IF NOT _DispatchValid() THEN
	RETURN;
ELSE
	_ClearTempString();
	ZaberCommand.stringval := Tc2_Standard.CONCAT(STR1 := ZaberConfiguration.sControllerRef, STR2 := ' ');
	ZaberCommand.stringval := Tc2_Standard.CONCAT(STR1 := ZaberCommand.stringval, STR2 := Base.F_GetFirstWordInString(sInput := SUPER^._iCommandConfiguration[ZaberStatus.ZaberMethodDispatch].P_CommandConfiguration.CommandDescription));
	ZaberCommand.stringval := Tc2_Standard.CONCAT(STR1 := ZaberCommand.stringval, STR2 := ' ');
	ZaberCommand.stringval := Tc2_Standard.CONCAT(STR1 := ZaberCommand.stringval, STR2 := USINT_TO_STRING(LockstepGroup));
	ZaberCommand.stringval := Tc2_Standard.CONCAT(STR1 := ZaberCommand.stringval, STR2 := ' ');
	ZaberCommand.stringval := Tc2_Standard.CONCAT(STR1 := ZaberCommand.stringval, STR2 := F_GetAllButFirstWord(sInput := SUPER^._iCommandConfiguration[ZaberStatus.ZaberMethodDispatch].P_CommandConfiguration.CommandDescription));
	
	IF iBufferSend <> 0 AND __QUERYINTERFACE(iBufferSend, testIBufferSend) THEN
		iBufferSend.AddObject(RefObject := ZaberCommand);
	END_IF
END_IF
END_METHOD

METHOD lockstep_move_abs
VAR_INPUT
	LockstepGroup	: USINT := 1; // The address of the lockstep group must be in the range 1 to lockstep.numgroups; lockstep.numgroups: the number of lockstep groupss; Valid Values: 0 to 2
	position		: UDINT := ZaberConfiguration.SetDynamics.Position;
	max_speed 		: UDINT := ZaberConfiguration.MaxDynamics.Velocity;
	accel			: UDINT := ZaberConfiguration.MaxDynamics.Accel;
END_VAR
IF ZaberStatus.ComponentStatus.iLastCommand <> 0 THEN
	ZaberStatus.ComponentStatus.iLastCommand.P_CommandStatus.LastCommandMessage := Base.F_GetLastWordInString(__POUNAME());
END_IF

IF NOT _DispatchValid() THEN
	RETURN;
ELSE
	_ClearTempString();
	ZaberCommand.stringval := Tc2_Standard.CONCAT(STR1 := ZaberConfiguration.sControllerRef, STR2 := ' ');
	ZaberCommand.stringval := Tc2_Standard.CONCAT(STR1 := ZaberCommand.stringval, STR2 := Base.F_GetFirstWordInString(sInput := SUPER^._iCommandConfiguration[ZaberStatus.ZaberMethodDispatch].P_CommandConfiguration.CommandDescription));
	ZaberCommand.stringval := Tc2_Standard.CONCAT(STR1 := ZaberCommand.stringval, STR2 := ' ');
	ZaberCommand.stringval := Tc2_Standard.CONCAT(STR1 := ZaberCommand.stringval, STR2 := USINT_TO_STRING(LockstepGroup));
	ZaberCommand.stringval := Tc2_Standard.CONCAT(STR1 := ZaberCommand.stringval, STR2 := ' ');
	ZaberCommand.stringval := Tc2_Standard.CONCAT(STR1 := ZaberCommand.stringval, STR2 := F_GetAllButFirstWord(sInput := SUPER^._iCommandConfiguration[ZaberStatus.ZaberMethodDispatch].P_CommandConfiguration.CommandDescription));
	ZaberCommand.stringval := Tc2_Standard.CONCAT(STR1 := ZaberCommand.stringval, STR2 := ' ');
	ZaberCommand.stringval := Tc2_Standard.CONCAT(STR1 := ZaberCommand.stringval, STR2 := UDINT_TO_STRING(position));
	ZaberCommand.stringval := Tc2_Standard.CONCAT(STR1 := ZaberCommand.stringval, STR2 := ' ');
	ZaberCommand.stringval := Tc2_Standard.CONCAT(STR1 := ZaberCommand.stringval, STR2 := UDINT_TO_STRING(max_speed));
	ZaberCommand.stringval := Tc2_Standard.CONCAT(STR1 := ZaberCommand.stringval, STR2 := ' ');
	ZaberCommand.stringval := Tc2_Standard.CONCAT(STR1 := ZaberCommand.stringval, STR2 := UDINT_TO_STRING(accel));
	
	IF iBufferSend <> 0 AND __QUERYINTERFACE(iBufferSend, testIBufferSend) THEN
		iBufferSend.AddObject(RefObject := ZaberCommand);
	END_IF
END_IF
END_METHOD

METHOD lockstep_move_rel
VAR_INPUT
	LockstepGroup	: USINT := 1; // The address of the lockstep group must be in the range 1 to lockstep.numgroups; lockstep.numgroups: the number of lockstep groupss; Valid Values: 0 to 2
	distance		: UDINT := ZaberConfiguration.SetDynamics.Position - ZaberStatus.Position;
	max_speed 		: UDINT := ZaberConfiguration.MaxDynamics.Velocity;
	accel			: UDINT := ZaberConfiguration.MaxDynamics.Accel;
END_VAR
IF ZaberStatus.ComponentStatus.iLastCommand <> 0 THEN
	ZaberStatus.ComponentStatus.iLastCommand.P_CommandStatus.LastCommandMessage := Base.F_GetLastWordInString(__POUNAME());
END_IF

IF NOT _DispatchValid() THEN
	RETURN;
ELSE
	_ClearTempString();
	ZaberCommand.stringval := Tc2_Standard.CONCAT(STR1 := ZaberConfiguration.sControllerRef, STR2 := ' ');
	ZaberCommand.stringval := Tc2_Standard.CONCAT(STR1 := ZaberCommand.stringval, STR2 := Base.F_GetFirstWordInString(sInput := SUPER^._iCommandConfiguration[ZaberStatus.ZaberMethodDispatch].P_CommandConfiguration.CommandDescription));
	ZaberCommand.stringval := Tc2_Standard.CONCAT(STR1 := ZaberCommand.stringval, STR2 := ' ');
	ZaberCommand.stringval := Tc2_Standard.CONCAT(STR1 := ZaberCommand.stringval, STR2 := USINT_TO_STRING(LockstepGroup));
	ZaberCommand.stringval := Tc2_Standard.CONCAT(STR1 := ZaberCommand.stringval, STR2 := ' ');
	ZaberCommand.stringval := Tc2_Standard.CONCAT(STR1 := ZaberCommand.stringval, STR2 := F_GetAllButFirstWord(sInput := SUPER^._iCommandConfiguration[ZaberStatus.ZaberMethodDispatch].P_CommandConfiguration.CommandDescription));
	ZaberCommand.stringval := Tc2_Standard.CONCAT(STR1 := ZaberCommand.stringval, STR2 := ' ');
	ZaberCommand.stringval := Tc2_Standard.CONCAT(STR1 := ZaberCommand.stringval, STR2 := UDINT_TO_STRING(distance));
	ZaberCommand.stringval := Tc2_Standard.CONCAT(STR1 := ZaberCommand.stringval, STR2 := ' ');
	ZaberCommand.stringval := Tc2_Standard.CONCAT(STR1 := ZaberCommand.stringval, STR2 := UDINT_TO_STRING(max_speed));
	ZaberCommand.stringval := Tc2_Standard.CONCAT(STR1 := ZaberCommand.stringval, STR2 := ' ');
	ZaberCommand.stringval := Tc2_Standard.CONCAT(STR1 := ZaberCommand.stringval, STR2 := UDINT_TO_STRING(accel));
	
	IF iBufferSend <> 0 AND __QUERYINTERFACE(iBufferSend, testIBufferSend) THEN
		iBufferSend.AddObject(RefObject := ZaberCommand);
	END_IF
END_IF
END_METHOD

METHOD lockstep_move_sin_stop
VAR_INPUT
	LockstepGroup	: USINT := 1; // The address of the lockstep group must be in the range 1 to lockstep.numgroups; lockstep.numgroups: the number of lockstep groupss; Valid Values: 0 to 2
END_VAR
IF ZaberStatus.ComponentStatus.iLastCommand <> 0 THEN
	ZaberStatus.ComponentStatus.iLastCommand.P_CommandStatus.LastCommandMessage := Base.F_GetLastWordInString(__POUNAME());
END_IF

IF NOT _DispatchValid() THEN
	RETURN;
ELSE
	_ClearTempString();
	ZaberCommand.stringval := Tc2_Standard.CONCAT(STR1 := ZaberConfiguration.sControllerRef, STR2 := ' ');
	ZaberCommand.stringval := Tc2_Standard.CONCAT(STR1 := ZaberCommand.stringval, STR2 := Base.F_GetFirstWordInString(sInput := SUPER^._iCommandConfiguration[ZaberStatus.ZaberMethodDispatch].P_CommandConfiguration.CommandDescription));
	ZaberCommand.stringval := Tc2_Standard.CONCAT(STR1 := ZaberCommand.stringval, STR2 := ' ');
	ZaberCommand.stringval := Tc2_Standard.CONCAT(STR1 := ZaberCommand.stringval, STR2 := USINT_TO_STRING(LockstepGroup));
	ZaberCommand.stringval := Tc2_Standard.CONCAT(STR1 := ZaberCommand.stringval, STR2 := ' ');
	ZaberCommand.stringval := Tc2_Standard.CONCAT(STR1 := ZaberCommand.stringval, STR2 := F_GetAllButFirstWord(sInput := SUPER^._iCommandConfiguration[ZaberStatus.ZaberMethodDispatch].P_CommandConfiguration.CommandDescription));
	
	IF iBufferSend <> 0 AND __QUERYINTERFACE(iBufferSend, testIBufferSend) THEN
		iBufferSend.AddObject(RefObject := ZaberCommand);
	END_IF
END_IF
END_METHOD

METHOD lockstep_move_stored
IF ZaberStatus.ComponentStatus.iLastCommand <> 0 THEN
	ZaberStatus.ComponentStatus.iLastCommand.P_CommandStatus.LastCommandMessage := Base.F_GetLastWordInString(__POUNAME());
END_IF

IF NOT _DispatchValid() THEN
	RETURN;
ELSE
	_BuildCommandStringNoArgs();
	
	IF iBufferSend <> 0 AND __QUERYINTERFACE(iBufferSend, testIBufferSend) THEN
		iBufferSend.AddObject(RefObject := ZaberCommand);
	END_IF
END_IF
END_METHOD

METHOD lockstep_move_vel
VAR_INPUT
	LockstepGroup	: USINT := 1; // The address of the lockstep group must be in the range 1 to lockstep.numgroups; lockstep.numgroups: the number of lockstep groupss; Valid Values: 0 to 2
	velocity		: DINT := ZaberConfiguration.SetDynamics.Velocity;
	accel			: UDINT := ZaberConfiguration.MaxDynamics.Accel;
END_VAR
IF ZaberStatus.ComponentStatus.iLastCommand <> 0 THEN
	ZaberStatus.ComponentStatus.iLastCommand.P_CommandStatus.LastCommandMessage := Base.F_GetLastWordInString(__POUNAME());
END_IF

IF NOT _DispatchValid() THEN
	RETURN;
ELSE
	_ClearTempString();
	ZaberCommand.stringval := Tc2_Standard.CONCAT(STR1 := ZaberConfiguration.sControllerRef, STR2 := ' ');
	ZaberCommand.stringval := Tc2_Standard.CONCAT(STR1 := ZaberCommand.stringval, STR2 := Base.F_GetFirstWordInString(sInput := SUPER^._iCommandConfiguration[ZaberStatus.ZaberMethodDispatch].P_CommandConfiguration.CommandDescription));
	ZaberCommand.stringval := Tc2_Standard.CONCAT(STR1 := ZaberCommand.stringval, STR2 := ' ');
	ZaberCommand.stringval := Tc2_Standard.CONCAT(STR1 := ZaberCommand.stringval, STR2 := USINT_TO_STRING(LockstepGroup));
	ZaberCommand.stringval := Tc2_Standard.CONCAT(STR1 := ZaberCommand.stringval, STR2 := ' ');
	ZaberCommand.stringval := Tc2_Standard.CONCAT(STR1 := ZaberCommand.stringval, STR2 := F_GetAllButFirstWord(sInput := SUPER^._iCommandConfiguration[ZaberStatus.ZaberMethodDispatch].P_CommandConfiguration.CommandDescription));
	ZaberCommand.stringval := Tc2_Standard.CONCAT(STR1 := ZaberCommand.stringval, STR2 := ' ');
	ZaberCommand.stringval := Tc2_Standard.CONCAT(STR1 := ZaberCommand.stringval, STR2 := UDINT_TO_STRING(velocity));
	ZaberCommand.stringval := Tc2_Standard.CONCAT(STR1 := ZaberCommand.stringval, STR2 := ' ');
	ZaberCommand.stringval := Tc2_Standard.CONCAT(STR1 := ZaberCommand.stringval, STR2 := UDINT_TO_STRING(accel));
	
	IF iBufferSend <> 0 AND __QUERYINTERFACE(iBufferSend, testIBufferSend) THEN
		iBufferSend.AddObject(RefObject := ZaberCommand);
	END_IF
END_IF
END_METHOD

METHOD lockstep_park
VAR_INPUT
	LockstepGroup	: USINT := 1; // The address of the lockstep group must be in the range 1 to lockstep.numgroups; lockstep.numgroups: the number of lockstep groupss; Valid Values: 0 to 2
END_VAR
IF ZaberStatus.ComponentStatus.iLastCommand <> 0 THEN
	ZaberStatus.ComponentStatus.iLastCommand.P_CommandStatus.LastCommandMessage := Base.F_GetLastWordInString(__POUNAME());
END_IF

IF NOT _DispatchValid() THEN
	RETURN;
ELSE
	_ClearTempString();
	ZaberCommand.stringval := Tc2_Standard.CONCAT(STR1 := ZaberConfiguration.sControllerRef, STR2 := ' ');
	ZaberCommand.stringval := Tc2_Standard.CONCAT(STR1 := ZaberCommand.stringval, STR2 := Base.F_GetFirstWordInString(sInput := SUPER^._iCommandConfiguration[ZaberStatus.ZaberMethodDispatch].P_CommandConfiguration.CommandDescription));
	ZaberCommand.stringval := Tc2_Standard.CONCAT(STR1 := ZaberCommand.stringval, STR2 := ' ');
	ZaberCommand.stringval := Tc2_Standard.CONCAT(STR1 := ZaberCommand.stringval, STR2 := USINT_TO_STRING(LockstepGroup));
	ZaberCommand.stringval := Tc2_Standard.CONCAT(STR1 := ZaberCommand.stringval, STR2 := ' ');
	ZaberCommand.stringval := Tc2_Standard.CONCAT(STR1 := ZaberCommand.stringval, STR2 := F_GetAllButFirstWord(sInput := SUPER^._iCommandConfiguration[ZaberStatus.ZaberMethodDispatch].P_CommandConfiguration.CommandDescription));
	
	IF iBufferSend <> 0 AND __QUERYINTERFACE(iBufferSend, testIBufferSend) THEN
		iBufferSend.AddObject(RefObject := ZaberCommand);
	END_IF
END_IF
END_METHOD

METHOD lockstep_print
VAR_INPUT
	LockstepGroup	: USINT := 1; // The address of the lockstep group must be in the range 1 to lockstep.numgroups; lockstep.numgroups: the number of lockstep groupss; Valid Values: 0 to 2
END_VAR
IF ZaberStatus.ComponentStatus.iLastCommand <> 0 THEN
	ZaberStatus.ComponentStatus.iLastCommand.P_CommandStatus.LastCommandMessage := Base.F_GetLastWordInString(__POUNAME());
END_IF

IF NOT _DispatchValid() THEN
	RETURN;
ELSE
	_ClearTempString();
	ZaberCommand.stringval := Tc2_Standard.CONCAT(STR1 := ZaberConfiguration.sControllerRef, STR2 := ' ');
	ZaberCommand.stringval := Tc2_Standard.CONCAT(STR1 := ZaberCommand.stringval, STR2 := Base.F_GetFirstWordInString(sInput := SUPER^._iCommandConfiguration[ZaberStatus.ZaberMethodDispatch].P_CommandConfiguration.CommandDescription));
	ZaberCommand.stringval := Tc2_Standard.CONCAT(STR1 := ZaberCommand.stringval, STR2 := ' ');
	ZaberCommand.stringval := Tc2_Standard.CONCAT(STR1 := ZaberCommand.stringval, STR2 := USINT_TO_STRING(LockstepGroup));
	ZaberCommand.stringval := Tc2_Standard.CONCAT(STR1 := ZaberCommand.stringval, STR2 := ' ');
	ZaberCommand.stringval := Tc2_Standard.CONCAT(STR1 := ZaberCommand.stringval, STR2 := F_GetAllButFirstWord(sInput := SUPER^._iCommandConfiguration[ZaberStatus.ZaberMethodDispatch].P_CommandConfiguration.CommandDescription));
	
	IF iBufferSend <> 0 AND __QUERYINTERFACE(iBufferSend, testIBufferSend) THEN
		iBufferSend.AddObject(RefObject := ZaberCommand);
	END_IF
END_IF
END_METHOD

METHOD lockstep_set_tolerance
VAR_INPUT
	LockstepGroup	: USINT := 1; // The address of the lockstep group must be in the range 1 to lockstep.numgroups; lockstep.numgroups: the number of lockstep groupss; Valid Values: 0 to 2
	Tolerance 		: UDINT := 150;
END_VAR
IF ZaberStatus.ComponentStatus.iLastCommand <> 0 THEN
	ZaberStatus.ComponentStatus.iLastCommand.P_CommandStatus.LastCommandMessage := Base.F_GetLastWordInString(__POUNAME());
END_IF

IF NOT _DispatchValid() THEN
	RETURN;
ELSE
	_ClearTempString();
	ZaberCommand.stringval := Tc2_Standard.CONCAT(STR1 := ZaberConfiguration.sControllerRef, STR2 := ' ');
	ZaberCommand.stringval := Tc2_Standard.CONCAT(STR1 := ZaberCommand.stringval, STR2 := UINT_TO_STRING(ZaberConfiguration.AxisRef));
	ZaberCommand.stringval := Tc2_Standard.CONCAT(STR1 := ZaberCommand.stringval, STR2 := ' ');
	ZaberCommand.stringval := Tc2_Standard.CONCAT(STR1 := ZaberCommand.stringval, STR2 := Base.F_GetFirstWordInString(sInput := SUPER^._iCommandConfiguration[ZaberStatus.ZaberMethodDispatch].P_CommandConfiguration.CommandDescription));
	ZaberCommand.stringval := Tc2_Standard.CONCAT(STR1 := ZaberCommand.stringval, STR2 := ' ');
	ZaberCommand.stringval := Tc2_Standard.CONCAT(STR1 := ZaberCommand.stringval, STR2 := USINT_TO_STRING(LockstepGroup));
	ZaberCommand.stringval := Tc2_Standard.CONCAT(STR1 := ZaberCommand.stringval, STR2 := ' ');
	ZaberCommand.stringval := Tc2_Standard.CONCAT(STR1 := ZaberCommand.stringval, STR2 := F_GetAllButFirstWord(sInput := SUPER^._iCommandConfiguration[ZaberStatus.ZaberMethodDispatch].P_CommandConfiguration.CommandDescription));
	ZaberCommand.stringval := Tc2_Standard.CONCAT(STR1 := ZaberCommand.stringval, STR2 := ' ');
	ZaberCommand.stringval := Tc2_Standard.CONCAT(STR1 := ZaberCommand.stringval, STR2 := UDINT_TO_STRING(Tolerance));;
	
	IF iBufferSend <> 0 AND __QUERYINTERFACE(iBufferSend, testIBufferSend) THEN
		iBufferSend.AddObject(RefObject := ZaberCommand);
	END_IF
END_IF
END_METHOD

METHOD lockstep_setup_disable
VAR_INPUT
	LockstepGroup	: USINT := 1; // The address of the lockstep group must be in the range 1 to lockstep.numgroups; lockstep.numgroups: the number of lockstep groupss; Valid Values: 0 to 2
END_VAR
IF ZaberStatus.ComponentStatus.iLastCommand <> 0 THEN
	ZaberStatus.ComponentStatus.iLastCommand.P_CommandStatus.LastCommandMessage := Base.F_GetLastWordInString(__POUNAME());
END_IF

IF NOT _DispatchValid() THEN
	RETURN;
ELSE
	_ClearTempString();
	ZaberCommand.stringval := Tc2_Standard.CONCAT(STR1 := ZaberConfiguration.sControllerRef, STR2 := ' ');
	ZaberCommand.stringval := Tc2_Standard.CONCAT(STR1 := ZaberCommand.stringval, STR2 := UINT_TO_STRING(ZaberConfiguration.AxisRef));
	ZaberCommand.stringval := Tc2_Standard.CONCAT(STR1 := ZaberCommand.stringval, STR2 := ' ');
	ZaberCommand.stringval := Tc2_Standard.CONCAT(STR1 := ZaberCommand.stringval, STR2 := Base.F_GetFirstWordInString(sInput := SUPER^._iCommandConfiguration[ZaberStatus.ZaberMethodDispatch].P_CommandConfiguration.CommandDescription));
	ZaberCommand.stringval := Tc2_Standard.CONCAT(STR1 := ZaberCommand.stringval, STR2 := ' ');
	ZaberCommand.stringval := Tc2_Standard.CONCAT(STR1 := ZaberCommand.stringval, STR2 := USINT_TO_STRING(LockstepGroup));
	ZaberCommand.stringval := Tc2_Standard.CONCAT(STR1 := ZaberCommand.stringval, STR2 := ' ');
	ZaberCommand.stringval := Tc2_Standard.CONCAT(STR1 := ZaberCommand.stringval, STR2 := F_GetAllButFirstWord(sInput := SUPER^._iCommandConfiguration[ZaberStatus.ZaberMethodDispatch].P_CommandConfiguration.CommandDescription));
	
	IF iBufferSend <> 0 AND __QUERYINTERFACE(iBufferSend, testIBufferSend) THEN
		iBufferSend.AddObject(RefObject := ZaberCommand);
	END_IF
END_IF
END_METHOD

METHOD lockstep_setup_enable
VAR_INPUT
	LockstepGroup	: USINT := 1; // The address of the lockstep group must be in the range 1 to lockstep.numgroups; lockstep.numgroups: the number of lockstep groupss; Valid Values: 0 to 2
	PrimaryAxis 	: USINT := 1;
	SecondaryAxis	: USINT := 2;
END_VAR
IF ZaberStatus.ComponentStatus.iLastCommand <> 0 THEN
	ZaberStatus.ComponentStatus.iLastCommand.P_CommandStatus.LastCommandMessage := Base.F_GetLastWordInString(__POUNAME());
END_IF

IF NOT _DispatchValid() THEN
	RETURN;
ELSE
	_ClearTempString();
	ZaberCommand.stringval := Tc2_Standard.CONCAT(STR1 := ZaberConfiguration.sControllerRef, STR2 := ' ');
	ZaberCommand.stringval := Tc2_Standard.CONCAT(STR1 := ZaberCommand.stringval, STR2 := UINT_TO_STRING(ZaberConfiguration.AxisRef));
	ZaberCommand.stringval := Tc2_Standard.CONCAT(STR1 := ZaberCommand.stringval, STR2 := ' ');
	ZaberCommand.stringval := Tc2_Standard.CONCAT(STR1 := ZaberCommand.stringval, STR2 := Base.F_GetFirstWordInString(sInput := SUPER^._iCommandConfiguration[ZaberStatus.ZaberMethodDispatch].P_CommandConfiguration.CommandDescription));
	ZaberCommand.stringval := Tc2_Standard.CONCAT(STR1 := ZaberCommand.stringval, STR2 := ' ');
	ZaberCommand.stringval := Tc2_Standard.CONCAT(STR1 := ZaberCommand.stringval, STR2 := USINT_TO_STRING(LockstepGroup));
	ZaberCommand.stringval := Tc2_Standard.CONCAT(STR1 := ZaberCommand.stringval, STR2 := ' ');
	ZaberCommand.stringval := Tc2_Standard.CONCAT(STR1 := ZaberCommand.stringval, STR2 := F_GetAllButFirstWord(sInput := SUPER^._iCommandConfiguration[ZaberStatus.ZaberMethodDispatch].P_CommandConfiguration.CommandDescription));
	ZaberCommand.stringval := Tc2_Standard.CONCAT(STR1 := ZaberCommand.stringval, STR2 := ' ');
	ZaberCommand.stringval := Tc2_Standard.CONCAT(STR1 := ZaberCommand.stringval, STR2 := USINT_TO_STRING(PrimaryAxis));
	ZaberCommand.stringval := Tc2_Standard.CONCAT(STR1 := ZaberCommand.stringval, STR2 := ' ');
	ZaberCommand.stringval := Tc2_Standard.CONCAT(STR1 := ZaberCommand.stringval, STR2 := USINT_TO_STRING(SecondaryAxis));
	
	IF iBufferSend <> 0 AND __QUERYINTERFACE(iBufferSend, testIBufferSend) THEN
		iBufferSend.AddObject(RefObject := ZaberCommand);
	END_IF
END_IF
END_METHOD

METHOD lockstep_stop
VAR_INPUT
	LockstepGroup	: USINT := 1; // The address of the lockstep group must be in the range 1 to lockstep.numgroups; lockstep.numgroups: the number of lockstep groupss; Valid Values: 0 to 2
END_VAR
IF ZaberStatus.ComponentStatus.iLastCommand <> 0 THEN
	ZaberStatus.ComponentStatus.iLastCommand.P_CommandStatus.LastCommandMessage := Base.F_GetLastWordInString(__POUNAME());
END_IF

IF NOT _DispatchValid() THEN
	RETURN;
ELSE
	_ClearTempString();
	ZaberCommand.stringval := Tc2_Standard.CONCAT(STR1 := ZaberConfiguration.sControllerRef, STR2 := ' ');
	ZaberCommand.stringval := Tc2_Standard.CONCAT(STR1 := ZaberCommand.stringval, STR2 := UINT_TO_STRING(ZaberConfiguration.AxisRef));
	ZaberCommand.stringval := Tc2_Standard.CONCAT(STR1 := ZaberCommand.stringval, STR2 := ' ');
	ZaberCommand.stringval := Tc2_Standard.CONCAT(STR1 := ZaberCommand.stringval, STR2 := Base.F_GetFirstWordInString(sInput := SUPER^._iCommandConfiguration[ZaberStatus.ZaberMethodDispatch].P_CommandConfiguration.CommandDescription));
	ZaberCommand.stringval := Tc2_Standard.CONCAT(STR1 := ZaberCommand.stringval, STR2 := ' ');
	ZaberCommand.stringval := Tc2_Standard.CONCAT(STR1 := ZaberCommand.stringval, STR2 := USINT_TO_STRING(LockstepGroup));
	ZaberCommand.stringval := Tc2_Standard.CONCAT(STR1 := ZaberCommand.stringval, STR2 := ' ');
	ZaberCommand.stringval := Tc2_Standard.CONCAT(STR1 := ZaberCommand.stringval, STR2 := F_GetAllButFirstWord(sInput := SUPER^._iCommandConfiguration[ZaberStatus.ZaberMethodDispatch].P_CommandConfiguration.CommandDescription));
	
	IF iBufferSend <> 0 AND __QUERYINTERFACE(iBufferSend, testIBufferSend) THEN
		iBufferSend.AddObject(RefObject := ZaberCommand);
	END_IF
END_IF
END_METHOD

METHOD lockstep_unpark
VAR_INPUT
	LockstepGroup	: USINT := 1; // The address of the lockstep group must be in the range 1 to lockstep.numgroups; lockstep.numgroups: the number of lockstep groupss; Valid Values: 0 to 2
END_VAR
IF ZaberStatus.ComponentStatus.iLastCommand <> 0 THEN
	ZaberStatus.ComponentStatus.iLastCommand.P_CommandStatus.LastCommandMessage := Base.F_GetLastWordInString(__POUNAME());
END_IF

IF NOT _DispatchValid() THEN
	RETURN;
ELSE
	_ClearTempString();
	ZaberCommand.stringval := Tc2_Standard.CONCAT(STR1 := ZaberConfiguration.sControllerRef, STR2 := ' ');
	ZaberCommand.stringval := Tc2_Standard.CONCAT(STR1 := ZaberCommand.stringval, STR2 := UINT_TO_STRING(ZaberConfiguration.AxisRef));
	ZaberCommand.stringval := Tc2_Standard.CONCAT(STR1 := ZaberCommand.stringval, STR2 := ' ');
	ZaberCommand.stringval := Tc2_Standard.CONCAT(STR1 := ZaberCommand.stringval, STR2 := Base.F_GetFirstWordInString(sInput := SUPER^._iCommandConfiguration[ZaberStatus.ZaberMethodDispatch].P_CommandConfiguration.CommandDescription));
	ZaberCommand.stringval := Tc2_Standard.CONCAT(STR1 := ZaberCommand.stringval, STR2 := ' ');
	ZaberCommand.stringval := Tc2_Standard.CONCAT(STR1 := ZaberCommand.stringval, STR2 := USINT_TO_STRING(LockstepGroup));
	ZaberCommand.stringval := Tc2_Standard.CONCAT(STR1 := ZaberCommand.stringval, STR2 := ' ');
	ZaberCommand.stringval := Tc2_Standard.CONCAT(STR1 := ZaberCommand.stringval, STR2 := F_GetAllButFirstWord(sInput := SUPER^._iCommandConfiguration[ZaberStatus.ZaberMethodDispatch].P_CommandConfiguration.CommandDescription));
	
	IF iBufferSend <> 0 AND __QUERYINTERFACE(iBufferSend, testIBufferSend) THEN
		iBufferSend.AddObject(RefObject := ZaberCommand);
	END_IF
END_IF
END_METHOD

METHOD move_index
IF ZaberStatus.ComponentStatus.iLastCommand <> 0 THEN
	ZaberStatus.ComponentStatus.iLastCommand.P_CommandStatus.LastCommandMessage := Base.F_GetLastWordInString(__POUNAME());
END_IF

IF NOT _DispatchValid() THEN
	RETURN;
ELSE
	_BuildCommandStringNoArgs();
	
	IF iBufferSend <> 0 AND __QUERYINTERFACE(iBufferSend, testIBufferSend) THEN
		iBufferSend.AddObject(RefObject := ZaberCommand);
	END_IF
END_IF
END_METHOD

METHOD move_rel
VAR_INPUT
	distance		: UDINT;
	max_speed 		: UDINT;
	accel			: UDINT;
END_VAR
IF ZaberStatus.ComponentStatus.iLastCommand <> 0 THEN
	ZaberStatus.ComponentStatus.iLastCommand.P_CommandStatus.LastCommandMessage := Base.F_GetLastWordInString(__POUNAME());
END_IF

IF NOT _DispatchValid() THEN
	RETURN;
ELSE
	_ClearTempString();
	ZaberCommand.stringval := Tc2_Standard.CONCAT(STR1 := ZaberConfiguration.sControllerRef, STR2 := ' ');
	ZaberCommand.stringval := Tc2_Standard.CONCAT(STR1 := ZaberCommand.stringval, STR2 := UINT_TO_STRING(ZaberConfiguration.AxisRef));
	ZaberCommand.stringval := Tc2_Standard.CONCAT(STR1 := ZaberCommand.stringval, STR2 := ' ');
	ZaberCommand.stringval := Tc2_Standard.CONCAT(STR1 := ZaberCommand.stringval, STR2 := SUPER^._iCommandConfiguration[ZaberStatus.ZaberMethodDispatch].P_CommandConfiguration.CommandDescription);
	ZaberCommand.stringval := Tc2_Standard.CONCAT(STR1 := ZaberCommand.stringval, STR2 := ' ');
	ZaberCommand.stringval := Tc2_Standard.CONCAT(STR1 := ZaberCommand.stringval, STR2 := UDINT_TO_STRING(distance));
	ZaberCommand.stringval := Tc2_Standard.CONCAT(STR1 := ZaberCommand.stringval, STR2 := ' ');
	ZaberCommand.stringval := Tc2_Standard.CONCAT(STR1 := ZaberCommand.stringval, STR2 := UDINT_TO_STRING(max_speed));
	ZaberCommand.stringval := Tc2_Standard.CONCAT(STR1 := ZaberCommand.stringval, STR2 := ' ');
	ZaberCommand.stringval := Tc2_Standard.CONCAT(STR1 := ZaberCommand.stringval, STR2 := UDINT_TO_STRING(accel));
		
	IF iBufferSend <> 0 AND __QUERYINTERFACE(iBufferSend, testIBufferSend) THEN
		iBufferSend.AddObject(RefObject := ZaberCommand);
	END_IF
END_IF
END_METHOD

METHOD move_sin_stop
IF ZaberStatus.ComponentStatus.iLastCommand <> 0 THEN
	ZaberStatus.ComponentStatus.iLastCommand.P_CommandStatus.LastCommandMessage := Base.F_GetLastWordInString(__POUNAME());
END_IF

IF NOT _DispatchValid() THEN
	RETURN;
ELSE
	_ClearTempString();
	ZaberCommand.stringval := Tc2_Standard.CONCAT(STR1 := ZaberConfiguration.sControllerRef, STR2 := ' ');
	ZaberCommand.stringval := Tc2_Standard.CONCAT(STR1 := ZaberCommand.stringval, STR2 := UINT_TO_STRING(ZaberConfiguration.AxisRef));
	ZaberCommand.stringval := Tc2_Standard.CONCAT(STR1 := ZaberCommand.stringval, STR2 := ' ');
	ZaberCommand.stringval := Tc2_Standard.CONCAT(STR1 := ZaberCommand.stringval, STR2 := SUPER^._iCommandConfiguration[ZaberStatus.ZaberMethodDispatch].P_CommandConfiguration.CommandDescription);
	
	IF iBufferSend <> 0 AND __QUERYINTERFACE(iBufferSend, testIBufferSend) THEN
		iBufferSend.AddObject(RefObject := ZaberCommand);
	END_IF
END_IF
END_METHOD

METHOD move_stored
IF ZaberStatus.ComponentStatus.iLastCommand <> 0 THEN
	ZaberStatus.ComponentStatus.iLastCommand.P_CommandStatus.LastCommandMessage := Base.F_GetLastWordInString(__POUNAME());
END_IF

IF NOT _DispatchValid() THEN
	RETURN;
ELSE
	_BuildCommandStringNoArgs();
	
	IF iBufferSend <> 0 AND __QUERYINTERFACE(iBufferSend, testIBufferSend) THEN
		iBufferSend.AddObject(RefObject := ZaberCommand);
	END_IF
END_IF
END_METHOD

METHOD pvt_buffer_erase
IF ZaberStatus.ComponentStatus.iLastCommand <> 0 THEN
	ZaberStatus.ComponentStatus.iLastCommand.P_CommandStatus.LastCommandMessage := Base.F_GetLastWordInString(__POUNAME());
END_IF

IF NOT _DispatchValid() THEN
	RETURN;
ELSE
	_BuildCommandStringNoArgs();
	
	IF iBufferSend <> 0 AND __QUERYINTERFACE(iBufferSend, testIBufferSend) THEN
		iBufferSend.AddObject(RefObject := ZaberCommand);
	END_IF
END_IF
END_METHOD

METHOD pvt_buffer_print
IF ZaberStatus.ComponentStatus.iLastCommand <> 0 THEN
	ZaberStatus.ComponentStatus.iLastCommand.P_CommandStatus.LastCommandMessage := Base.F_GetLastWordInString(__POUNAME());
END_IF

IF NOT _DispatchValid() THEN
	RETURN;
ELSE
	_BuildCommandStringNoArgs();
	
	IF iBufferSend <> 0 AND __QUERYINTERFACE(iBufferSend, testIBufferSend) THEN
		iBufferSend.AddObject(RefObject := ZaberCommand);
	END_IF
END_IF
END_METHOD

METHOD pvt_call
IF ZaberStatus.ComponentStatus.iLastCommand <> 0 THEN
	ZaberStatus.ComponentStatus.iLastCommand.P_CommandStatus.LastCommandMessage := Base.F_GetLastWordInString(__POUNAME());
END_IF

IF NOT _DispatchValid() THEN
	RETURN;
ELSE
	_BuildCommandStringNoArgs();
	
	IF iBufferSend <> 0 AND __QUERYINTERFACE(iBufferSend, testIBufferSend) THEN
		iBufferSend.AddObject(RefObject := ZaberCommand);
	END_IF
END_IF
END_METHOD

METHOD pvt_fifo
IF ZaberStatus.ComponentStatus.iLastCommand <> 0 THEN
	ZaberStatus.ComponentStatus.iLastCommand.P_CommandStatus.LastCommandMessage := Base.F_GetLastWordInString(__POUNAME());
END_IF

IF NOT _DispatchValid() THEN
	RETURN;
ELSE
	_BuildCommandStringNoArgs();
	
	IF iBufferSend <> 0 AND __QUERYINTERFACE(iBufferSend, testIBufferSend) THEN
		iBufferSend.AddObject(RefObject := ZaberCommand);
	END_IF
END_IF
END_METHOD

METHOD pvt_info
IF ZaberStatus.ComponentStatus.iLastCommand <> 0 THEN
	ZaberStatus.ComponentStatus.iLastCommand.P_CommandStatus.LastCommandMessage := Base.F_GetLastWordInString(__POUNAME());
END_IF

IF NOT _DispatchValid() THEN
	RETURN;
ELSE
	_BuildCommandStringNoArgs();
	
	IF iBufferSend <> 0 AND __QUERYINTERFACE(iBufferSend, testIBufferSend) THEN
		iBufferSend.AddObject(RefObject := ZaberCommand);
	END_IF
END_IF
END_METHOD

METHOD pvt_io_cancel_schedule
IF ZaberStatus.ComponentStatus.iLastCommand <> 0 THEN
	ZaberStatus.ComponentStatus.iLastCommand.P_CommandStatus.LastCommandMessage := Base.F_GetLastWordInString(__POUNAME());
END_IF

IF NOT _DispatchValid() THEN
	RETURN;
ELSE
	_BuildCommandStringNoArgs();
	
	IF iBufferSend <> 0 AND __QUERYINTERFACE(iBufferSend, testIBufferSend) THEN
		iBufferSend.AddObject(RefObject := ZaberCommand);
	END_IF
END_IF
END_METHOD

METHOD pvt_io_set_ao
IF ZaberStatus.ComponentStatus.iLastCommand <> 0 THEN
	ZaberStatus.ComponentStatus.iLastCommand.P_CommandStatus.LastCommandMessage := Base.F_GetLastWordInString(__POUNAME());
END_IF

IF NOT _DispatchValid() THEN
	RETURN;
ELSE
	_BuildCommandStringNoArgs();
	
	IF iBufferSend <> 0 AND __QUERYINTERFACE(iBufferSend, testIBufferSend) THEN
		iBufferSend.AddObject(RefObject := ZaberCommand);
	END_IF
END_IF
END_METHOD

METHOD pvt_io_set_ao_schedule
IF ZaberStatus.ComponentStatus.iLastCommand <> 0 THEN
	ZaberStatus.ComponentStatus.iLastCommand.P_CommandStatus.LastCommandMessage := Base.F_GetLastWordInString(__POUNAME());
END_IF

IF NOT _DispatchValid() THEN
	RETURN;
ELSE
	_BuildCommandStringNoArgs();
	
	IF iBufferSend <> 0 AND __QUERYINTERFACE(iBufferSend, testIBufferSend) THEN
		iBufferSend.AddObject(RefObject := ZaberCommand);
	END_IF
END_IF
END_METHOD

METHOD pvt_io_set_do
IF ZaberStatus.ComponentStatus.iLastCommand <> 0 THEN
	ZaberStatus.ComponentStatus.iLastCommand.P_CommandStatus.LastCommandMessage := Base.F_GetLastWordInString(__POUNAME());
END_IF

IF NOT _DispatchValid() THEN
	RETURN;
ELSE
	_BuildCommandStringNoArgs();
	
	IF iBufferSend <> 0 AND __QUERYINTERFACE(iBufferSend, testIBufferSend) THEN
		iBufferSend.AddObject(RefObject := ZaberCommand);
	END_IF
END_IF
END_METHOD

METHOD pvt_io_set_do_schedule
IF ZaberStatus.ComponentStatus.iLastCommand <> 0 THEN
	ZaberStatus.ComponentStatus.iLastCommand.P_CommandStatus.LastCommandMessage := Base.F_GetLastWordInString(__POUNAME());
END_IF

IF NOT _DispatchValid() THEN
	RETURN;
ELSE
	_BuildCommandStringNoArgs();
	
	IF iBufferSend <> 0 AND __QUERYINTERFACE(iBufferSend, testIBufferSend) THEN
		iBufferSend.AddObject(RefObject := ZaberCommand);
	END_IF
END_IF
END_METHOD

METHOD pvt_point
IF ZaberStatus.ComponentStatus.iLastCommand <> 0 THEN
	ZaberStatus.ComponentStatus.iLastCommand.P_CommandStatus.LastCommandMessage := Base.F_GetLastWordInString(__POUNAME());
END_IF

IF NOT _DispatchValid() THEN
	RETURN;
ELSE
	_BuildCommandStringNoArgs();
	
	IF iBufferSend <> 0 AND __QUERYINTERFACE(iBufferSend, testIBufferSend) THEN
		iBufferSend.AddObject(RefObject := ZaberCommand);
	END_IF
END_IF
END_METHOD

METHOD pvt_setup_disable
IF ZaberStatus.ComponentStatus.iLastCommand <> 0 THEN
	ZaberStatus.ComponentStatus.iLastCommand.P_CommandStatus.LastCommandMessage := Base.F_GetLastWordInString(__POUNAME());
END_IF

IF NOT _DispatchValid() THEN
	RETURN;
ELSE
	_BuildCommandStringNoArgs();
	
	IF iBufferSend <> 0 AND __QUERYINTERFACE(iBufferSend, testIBufferSend) THEN
		iBufferSend.AddObject(RefObject := ZaberCommand);
	END_IF
END_IF
END_METHOD

METHOD pvt_setup_live
IF ZaberStatus.ComponentStatus.iLastCommand <> 0 THEN
	ZaberStatus.ComponentStatus.iLastCommand.P_CommandStatus.LastCommandMessage := Base.F_GetLastWordInString(__POUNAME());
END_IF

IF NOT _DispatchValid() THEN
	RETURN;
ELSE
	_BuildCommandStringNoArgs();
	
	IF iBufferSend <> 0 AND __QUERYINTERFACE(iBufferSend, testIBufferSend) THEN
		iBufferSend.AddObject(RefObject := ZaberCommand);
	END_IF
END_IF
END_METHOD

METHOD pvt_setup_store
IF ZaberStatus.ComponentStatus.iLastCommand <> 0 THEN
	ZaberStatus.ComponentStatus.iLastCommand.P_CommandStatus.LastCommandMessage := Base.F_GetLastWordInString(__POUNAME());
END_IF

IF NOT _DispatchValid() THEN
	RETURN;
ELSE
	_BuildCommandStringNoArgs();
	
	IF iBufferSend <> 0 AND __QUERYINTERFACE(iBufferSend, testIBufferSend) THEN
		iBufferSend.AddObject(RefObject := ZaberCommand);
	END_IF
END_IF
END_METHOD

METHOD scope_add
IF ZaberStatus.ComponentStatus.iLastCommand <> 0 THEN
	ZaberStatus.ComponentStatus.iLastCommand.P_CommandStatus.LastCommandMessage := Base.F_GetLastWordInString(__POUNAME());
END_IF

IF NOT _DispatchValid() THEN
	RETURN;
ELSE
	_BuildCommandStringNoArgs();
	
	IF iBufferSend <> 0 AND __QUERYINTERFACE(iBufferSend, testIBufferSend) THEN
		iBufferSend.AddObject(RefObject := ZaberCommand);
	END_IF
END_IF
END_METHOD

METHOD scope_add_io_ai
IF ZaberStatus.ComponentStatus.iLastCommand <> 0 THEN
	ZaberStatus.ComponentStatus.iLastCommand.P_CommandStatus.LastCommandMessage := Base.F_GetLastWordInString(__POUNAME());
END_IF

IF NOT _DispatchValid() THEN
	RETURN;
ELSE
	_BuildCommandStringNoArgs();
	
	IF iBufferSend <> 0 AND __QUERYINTERFACE(iBufferSend, testIBufferSend) THEN
		iBufferSend.AddObject(RefObject := ZaberCommand);
	END_IF
END_IF
END_METHOD

METHOD scope_add_io_ao
IF ZaberStatus.ComponentStatus.iLastCommand <> 0 THEN
	ZaberStatus.ComponentStatus.iLastCommand.P_CommandStatus.LastCommandMessage := Base.F_GetLastWordInString(__POUNAME());
END_IF

IF NOT _DispatchValid() THEN
	RETURN;
ELSE
	_BuildCommandStringNoArgs();
	
	IF iBufferSend <> 0 AND __QUERYINTERFACE(iBufferSend, testIBufferSend) THEN
		iBufferSend.AddObject(RefObject := ZaberCommand);
	END_IF
END_IF
END_METHOD

METHOD scope_add_io_di
IF ZaberStatus.ComponentStatus.iLastCommand <> 0 THEN
	ZaberStatus.ComponentStatus.iLastCommand.P_CommandStatus.LastCommandMessage := Base.F_GetLastWordInString(__POUNAME());
END_IF

IF NOT _DispatchValid() THEN
	RETURN;
ELSE
	_BuildCommandStringNoArgs();
	
	IF iBufferSend <> 0 AND __QUERYINTERFACE(iBufferSend, testIBufferSend) THEN
		iBufferSend.AddObject(RefObject := ZaberCommand);
	END_IF
END_IF
END_METHOD

METHOD scope_add_io_do
IF ZaberStatus.ComponentStatus.iLastCommand <> 0 THEN
	ZaberStatus.ComponentStatus.iLastCommand.P_CommandStatus.LastCommandMessage := Base.F_GetLastWordInString(__POUNAME());
END_IF

IF NOT _DispatchValid() THEN
	RETURN;
ELSE
	_BuildCommandStringNoArgs();
	
	IF iBufferSend <> 0 AND __QUERYINTERFACE(iBufferSend, testIBufferSend) THEN
		iBufferSend.AddObject(RefObject := ZaberCommand);
	END_IF
END_IF
END_METHOD

METHOD scope_start
IF ZaberStatus.ComponentStatus.iLastCommand <> 0 THEN
	ZaberStatus.ComponentStatus.iLastCommand.P_CommandStatus.LastCommandMessage := Base.F_GetLastWordInString(__POUNAME());
END_IF

IF NOT _DispatchValid() THEN
	RETURN;
ELSE
	_BuildCommandStringNoArgs();
	
	IF iBufferSend <> 0 AND __QUERYINTERFACE(iBufferSend, testIBufferSend) THEN
		iBufferSend.AddObject(RefObject := ZaberCommand);
	END_IF
END_IF
END_METHOD

METHOD set_accel
IF ZaberStatus.ComponentStatus.iLastCommand <> 0 THEN
	ZaberStatus.ComponentStatus.iLastCommand.P_CommandStatus.LastCommandMessage := Base.F_GetLastWordInString(__POUNAME());
END_IF

IF NOT _DispatchValid() THEN
	RETURN;
ELSE
	_BuildCommandStringNoArgs();
	
	IF iBufferSend <> 0 AND __QUERYINTERFACE(iBufferSend, testIBufferSend) THEN
		iBufferSend.AddObject(RefObject := ZaberCommand);
	END_IF
END_IF
END_METHOD

METHOD set_autodetect_coil_mode
IF ZaberStatus.ComponentStatus.iLastCommand <> 0 THEN
	ZaberStatus.ComponentStatus.iLastCommand.P_CommandStatus.LastCommandMessage := Base.F_GetLastWordInString(__POUNAME());
END_IF

IF NOT _DispatchValid() THEN
	RETURN;
ELSE
	_BuildCommandStringNoArgs();
	
	IF iBufferSend <> 0 AND __QUERYINTERFACE(iBufferSend, testIBufferSend) THEN
		iBufferSend.AddObject(RefObject := ZaberCommand);
	END_IF
END_IF
END_METHOD

METHOD set_calibration_type
IF ZaberStatus.ComponentStatus.iLastCommand <> 0 THEN
	ZaberStatus.ComponentStatus.iLastCommand.P_CommandStatus.LastCommandMessage := Base.F_GetLastWordInString(__POUNAME());
END_IF

IF NOT _DispatchValid() THEN
	RETURN;
ELSE
	_BuildCommandStringNoArgs();
	
	IF iBufferSend <> 0 AND __QUERYINTERFACE(iBufferSend, testIBufferSend) THEN
		iBufferSend.AddObject(RefObject := ZaberCommand);
	END_IF
END_IF
END_METHOD

METHOD set_comm_address
IF ZaberStatus.ComponentStatus.iLastCommand <> 0 THEN
	ZaberStatus.ComponentStatus.iLastCommand.P_CommandStatus.LastCommandMessage := Base.F_GetLastWordInString(__POUNAME());
END_IF

IF NOT _DispatchValid() THEN
	RETURN;
ELSE
	_BuildCommandStringNoArgs();
	
	IF iBufferSend <> 0 AND __QUERYINTERFACE(iBufferSend, testIBufferSend) THEN
		iBufferSend.AddObject(RefObject := ZaberCommand);
	END_IF
END_IF
END_METHOD

METHOD set_comm_alert
IF ZaberStatus.ComponentStatus.iLastCommand <> 0 THEN
	ZaberStatus.ComponentStatus.iLastCommand.P_CommandStatus.LastCommandMessage := Base.F_GetLastWordInString(__POUNAME());
END_IF

IF NOT _DispatchValid() THEN
	RETURN;
ELSE
	_BuildCommandStringNoArgs();
	
	IF iBufferSend <> 0 AND __QUERYINTERFACE(iBufferSend, testIBufferSend) THEN
		iBufferSend.AddObject(RefObject := ZaberCommand);
	END_IF
END_IF
END_METHOD

METHOD set_comm_command_packets_max
IF ZaberStatus.ComponentStatus.iLastCommand <> 0 THEN
	ZaberStatus.ComponentStatus.iLastCommand.P_CommandStatus.LastCommandMessage := Base.F_GetLastWordInString(__POUNAME());
END_IF

IF NOT _DispatchValid() THEN
	RETURN;
ELSE
	_BuildCommandStringNoArgs();
	
	IF iBufferSend <> 0 AND __QUERYINTERFACE(iBufferSend, testIBufferSend) THEN
		iBufferSend.AddObject(RefObject := ZaberCommand);
	END_IF
END_IF
END_METHOD

METHOD set_comm_en_ipv4_address
IF ZaberStatus.ComponentStatus.iLastCommand <> 0 THEN
	ZaberStatus.ComponentStatus.iLastCommand.P_CommandStatus.LastCommandMessage := Base.F_GetLastWordInString(__POUNAME());
END_IF

IF NOT _DispatchValid() THEN
	RETURN;
ELSE
	_BuildCommandStringNoArgs();
	
	IF iBufferSend <> 0 AND __QUERYINTERFACE(iBufferSend, testIBufferSend) THEN
		iBufferSend.AddObject(RefObject := ZaberCommand);
	END_IF
END_IF
END_METHOD

METHOD set_comm_en_ipv4_dhcp_enabled
IF ZaberStatus.ComponentStatus.iLastCommand <> 0 THEN
	ZaberStatus.ComponentStatus.iLastCommand.P_CommandStatus.LastCommandMessage := Base.F_GetLastWordInString(__POUNAME());
END_IF

IF NOT _DispatchValid() THEN
	RETURN;
ELSE
	_BuildCommandStringNoArgs();
	
	IF iBufferSend <> 0 AND __QUERYINTERFACE(iBufferSend, testIBufferSend) THEN
		iBufferSend.AddObject(RefObject := ZaberCommand);
	END_IF
END_IF
END_METHOD

METHOD set_comm_en_ipv4_gateway
IF ZaberStatus.ComponentStatus.iLastCommand <> 0 THEN
	ZaberStatus.ComponentStatus.iLastCommand.P_CommandStatus.LastCommandMessage := Base.F_GetLastWordInString(__POUNAME());
END_IF

IF NOT _DispatchValid() THEN
	RETURN;
ELSE
	_BuildCommandStringNoArgs();
	
	IF iBufferSend <> 0 AND __QUERYINTERFACE(iBufferSend, testIBufferSend) THEN
		iBufferSend.AddObject(RefObject := ZaberCommand);
	END_IF
END_IF
END_METHOD

METHOD set_comm_en_ipv4_netmask
IF ZaberStatus.ComponentStatus.iLastCommand <> 0 THEN
	ZaberStatus.ComponentStatus.iLastCommand.P_CommandStatus.LastCommandMessage := Base.F_GetLastWordInString(__POUNAME());
END_IF

IF NOT _DispatchValid() THEN
	RETURN;
ELSE
	_BuildCommandStringNoArgs();
	
	IF iBufferSend <> 0 AND __QUERYINTERFACE(iBufferSend, testIBufferSend) THEN
		iBufferSend.AddObject(RefObject := ZaberCommand);
	END_IF
END_IF
END_METHOD

METHOD set_comm_en_mac
IF ZaberStatus.ComponentStatus.iLastCommand <> 0 THEN
	ZaberStatus.ComponentStatus.iLastCommand.P_CommandStatus.LastCommandMessage := Base.F_GetLastWordInString(__POUNAME());
END_IF

IF NOT _DispatchValid() THEN
	RETURN;
ELSE
	_BuildCommandStringNoArgs();
	
	IF iBufferSend <> 0 AND __QUERYINTERFACE(iBufferSend, testIBufferSend) THEN
		iBufferSend.AddObject(RefObject := ZaberCommand);
	END_IF
END_IF
END_METHOD

METHOD set_comm_en_mdns_enable
IF ZaberStatus.ComponentStatus.iLastCommand <> 0 THEN
	ZaberStatus.ComponentStatus.iLastCommand.P_CommandStatus.LastCommandMessage := Base.F_GetLastWordInString(__POUNAME());
END_IF

IF NOT _DispatchValid() THEN
	RETURN;
ELSE
	_BuildCommandStringNoArgs();
	
	IF iBufferSend <> 0 AND __QUERYINTERFACE(iBufferSend, testIBufferSend) THEN
		iBufferSend.AddObject(RefObject := ZaberCommand);
	END_IF
END_IF
END_METHOD

METHOD set_comm_next_owner
IF ZaberStatus.ComponentStatus.iLastCommand <> 0 THEN
	ZaberStatus.ComponentStatus.iLastCommand.P_CommandStatus.LastCommandMessage := Base.F_GetLastWordInString(__POUNAME());
END_IF

IF NOT _DispatchValid() THEN
	RETURN;
ELSE
	_BuildCommandStringNoArgs();
	
	IF iBufferSend <> 0 AND __QUERYINTERFACE(iBufferSend, testIBufferSend) THEN
		iBufferSend.AddObject(RefObject := ZaberCommand);
	END_IF
END_IF
END_METHOD

METHOD set_comm_packet_size_max
IF ZaberStatus.ComponentStatus.iLastCommand <> 0 THEN
	ZaberStatus.ComponentStatus.iLastCommand.P_CommandStatus.LastCommandMessage := Base.F_GetLastWordInString(__POUNAME());
END_IF

IF NOT _DispatchValid() THEN
	RETURN;
ELSE
	_BuildCommandStringNoArgs();
	
	IF iBufferSend <> 0 AND __QUERYINTERFACE(iBufferSend, testIBufferSend) THEN
		iBufferSend.AddObject(RefObject := ZaberCommand);
	END_IF
END_IF
END_METHOD

METHOD set_comm_protocol
IF ZaberStatus.ComponentStatus.iLastCommand <> 0 THEN
	ZaberStatus.ComponentStatus.iLastCommand.P_CommandStatus.LastCommandMessage := Base.F_GetLastWordInString(__POUNAME());
END_IF

IF NOT _DispatchValid() THEN
	RETURN;
ELSE
	_BuildCommandStringNoArgs();
	
	IF iBufferSend <> 0 AND __QUERYINTERFACE(iBufferSend, testIBufferSend) THEN
		iBufferSend.AddObject(RefObject := ZaberCommand);
	END_IF
END_IF
END_METHOD

METHOD set_comm_rs232_baud
IF ZaberStatus.ComponentStatus.iLastCommand <> 0 THEN
	ZaberStatus.ComponentStatus.iLastCommand.P_CommandStatus.LastCommandMessage := Base.F_GetLastWordInString(__POUNAME());
END_IF

IF NOT _DispatchValid() THEN
	RETURN;
ELSE
	_BuildCommandStringNoArgs();
	
	IF iBufferSend <> 0 AND __QUERYINTERFACE(iBufferSend, testIBufferSend) THEN
		iBufferSend.AddObject(RefObject := ZaberCommand);
	END_IF
END_IF
END_METHOD

METHOD set_comm_word_size_max
IF ZaberStatus.ComponentStatus.iLastCommand <> 0 THEN
	ZaberStatus.ComponentStatus.iLastCommand.P_CommandStatus.LastCommandMessage := Base.F_GetLastWordInString(__POUNAME());
END_IF

IF NOT _DispatchValid() THEN
	RETURN;
ELSE
	_BuildCommandStringNoArgs();
	
	IF iBufferSend <> 0 AND __QUERYINTERFACE(iBufferSend, testIBufferSend) THEN
		iBufferSend.AddObject(RefObject := ZaberCommand);
	END_IF
END_IF
END_METHOD

METHOD set_driver_current_approach
IF ZaberStatus.ComponentStatus.iLastCommand <> 0 THEN
	ZaberStatus.ComponentStatus.iLastCommand.P_CommandStatus.LastCommandMessage := Base.F_GetLastWordInString(__POUNAME());
END_IF

IF NOT _DispatchValid() THEN
	RETURN;
ELSE
	_BuildCommandStringNoArgs();
	
	IF iBufferSend <> 0 AND __QUERYINTERFACE(iBufferSend, testIBufferSend) THEN
		iBufferSend.AddObject(RefObject := ZaberCommand);
	END_IF
END_IF
END_METHOD

METHOD set_driver_current_hold
IF ZaberStatus.ComponentStatus.iLastCommand <> 0 THEN
	ZaberStatus.ComponentStatus.iLastCommand.P_CommandStatus.LastCommandMessage := Base.F_GetLastWordInString(__POUNAME());
END_IF

IF NOT _DispatchValid() THEN
	RETURN;
ELSE
	_BuildCommandStringNoArgs();
	
	IF iBufferSend <> 0 AND __QUERYINTERFACE(iBufferSend, testIBufferSend) THEN
		iBufferSend.AddObject(RefObject := ZaberCommand);
	END_IF
END_IF
END_METHOD

METHOD set_driver_current_max
IF ZaberStatus.ComponentStatus.iLastCommand <> 0 THEN
	ZaberStatus.ComponentStatus.iLastCommand.P_CommandStatus.LastCommandMessage := Base.F_GetLastWordInString(__POUNAME());
END_IF

IF NOT _DispatchValid() THEN
	RETURN;
ELSE
	_BuildCommandStringNoArgs();
	
	IF iBufferSend <> 0 AND __QUERYINTERFACE(iBufferSend, testIBufferSend) THEN
		iBufferSend.AddObject(RefObject := ZaberCommand);
	END_IF
END_IF
END_METHOD

METHOD set_driver_current_run
IF ZaberStatus.ComponentStatus.iLastCommand <> 0 THEN
	ZaberStatus.ComponentStatus.iLastCommand.P_CommandStatus.LastCommandMessage := Base.F_GetLastWordInString(__POUNAME());
END_IF

IF NOT _DispatchValid() THEN
	RETURN;
ELSE
	_BuildCommandStringNoArgs();
	
	IF iBufferSend <> 0 AND __QUERYINTERFACE(iBufferSend, testIBufferSend) THEN
		iBufferSend.AddObject(RefObject := ZaberCommand);
	END_IF
END_IF
END_METHOD

METHOD set_driver_enable_mode
IF ZaberStatus.ComponentStatus.iLastCommand <> 0 THEN
	ZaberStatus.ComponentStatus.iLastCommand.P_CommandStatus.LastCommandMessage := Base.F_GetLastWordInString(__POUNAME());
END_IF

IF NOT _DispatchValid() THEN
	RETURN;
ELSE
	_BuildCommandStringNoArgs();
	
	IF iBufferSend <> 0 AND __QUERYINTERFACE(iBufferSend, testIBufferSend) THEN
		iBufferSend.AddObject(RefObject := ZaberCommand);
	END_IF
END_IF
END_METHOD

METHOD set_driver_enabled
IF ZaberStatus.ComponentStatus.iLastCommand <> 0 THEN
	ZaberStatus.ComponentStatus.iLastCommand.P_CommandStatus.LastCommandMessage := Base.F_GetLastWordInString(__POUNAME());
END_IF

IF NOT _DispatchValid() THEN
	RETURN;
ELSE
	_BuildCommandStringNoArgs();
	
	IF iBufferSend <> 0 AND __QUERYINTERFACE(iBufferSend, testIBufferSend) THEN
		iBufferSend.AddObject(RefObject := ZaberCommand);
	END_IF
END_IF
END_METHOD

METHOD set_driver_temperature
IF ZaberStatus.ComponentStatus.iLastCommand <> 0 THEN
	ZaberStatus.ComponentStatus.iLastCommand.P_CommandStatus.LastCommandMessage := Base.F_GetLastWordInString(__POUNAME());
END_IF

IF NOT _DispatchValid() THEN
	RETURN;
ELSE
	_BuildCommandStringNoArgs();
	
	IF iBufferSend <> 0 AND __QUERYINTERFACE(iBufferSend, testIBufferSend) THEN
		iBufferSend.AddObject(RefObject := ZaberCommand);
	END_IF
END_IF
END_METHOD

METHOD set_get_settings_max
IF ZaberStatus.ComponentStatus.iLastCommand <> 0 THEN
	ZaberStatus.ComponentStatus.iLastCommand.P_CommandStatus.LastCommandMessage := Base.F_GetLastWordInString(__POUNAME());
END_IF

IF NOT _DispatchValid() THEN
	RETURN;
ELSE
	_BuildCommandStringNoArgs();
	
	IF iBufferSend <> 0 AND __QUERYINTERFACE(iBufferSend, testIBufferSend) THEN
		iBufferSend.AddObject(RefObject := ZaberCommand);
	END_IF
END_IF
END_METHOD

METHOD set_ictrl_advance_a
IF ZaberStatus.ComponentStatus.iLastCommand <> 0 THEN
	ZaberStatus.ComponentStatus.iLastCommand.P_CommandStatus.LastCommandMessage := Base.F_GetLastWordInString(__POUNAME());
END_IF

IF NOT _DispatchValid() THEN
	RETURN;
ELSE
	_BuildCommandStringNoArgs();
	
	IF iBufferSend <> 0 AND __QUERYINTERFACE(iBufferSend, testIBufferSend) THEN
		iBufferSend.AddObject(RefObject := ZaberCommand);
	END_IF
END_IF
END_METHOD

METHOD set_ictrl_advance_offset
IF ZaberStatus.ComponentStatus.iLastCommand <> 0 THEN
	ZaberStatus.ComponentStatus.iLastCommand.P_CommandStatus.LastCommandMessage := Base.F_GetLastWordInString(__POUNAME());
END_IF

IF NOT _DispatchValid() THEN
	RETURN;
ELSE
	_BuildCommandStringNoArgs();
	
	IF iBufferSend <> 0 AND __QUERYINTERFACE(iBufferSend, testIBufferSend) THEN
		iBufferSend.AddObject(RefObject := ZaberCommand);
	END_IF
END_IF
END_METHOD

METHOD set_ictrl_afcff_inductance
IF ZaberStatus.ComponentStatus.iLastCommand <> 0 THEN
	ZaberStatus.ComponentStatus.iLastCommand.P_CommandStatus.LastCommandMessage := Base.F_GetLastWordInString(__POUNAME());
END_IF

IF NOT _DispatchValid() THEN
	RETURN;
ELSE
	_BuildCommandStringNoArgs();
	
	IF iBufferSend <> 0 AND __QUERYINTERFACE(iBufferSend, testIBufferSend) THEN
		iBufferSend.AddObject(RefObject := ZaberCommand);
	END_IF
END_IF
END_METHOD

METHOD set_ictrl_afcff_ke
IF ZaberStatus.ComponentStatus.iLastCommand <> 0 THEN
	ZaberStatus.ComponentStatus.iLastCommand.P_CommandStatus.LastCommandMessage := Base.F_GetLastWordInString(__POUNAME());
END_IF

IF NOT _DispatchValid() THEN
	RETURN;
ELSE
	_BuildCommandStringNoArgs();
	
	IF iBufferSend <> 0 AND __QUERYINTERFACE(iBufferSend, testIBufferSend) THEN
		iBufferSend.AddObject(RefObject := ZaberCommand);
	END_IF
END_IF
END_METHOD

METHOD set_ictrl_afcff_ki
IF ZaberStatus.ComponentStatus.iLastCommand <> 0 THEN
	ZaberStatus.ComponentStatus.iLastCommand.P_CommandStatus.LastCommandMessage := Base.F_GetLastWordInString(__POUNAME());
END_IF

IF NOT _DispatchValid() THEN
	RETURN;
ELSE
	_BuildCommandStringNoArgs();
	
	IF iBufferSend <> 0 AND __QUERYINTERFACE(iBufferSend, testIBufferSend) THEN
		iBufferSend.AddObject(RefObject := ZaberCommand);
	END_IF
END_IF
END_METHOD

METHOD set_ictrl_afcff_max
IF ZaberStatus.ComponentStatus.iLastCommand <> 0 THEN
	ZaberStatus.ComponentStatus.iLastCommand.P_CommandStatus.LastCommandMessage := Base.F_GetLastWordInString(__POUNAME());
END_IF

IF NOT _DispatchValid() THEN
	RETURN;
ELSE
	_BuildCommandStringNoArgs();
	
	IF iBufferSend <> 0 AND __QUERYINTERFACE(iBufferSend, testIBufferSend) THEN
		iBufferSend.AddObject(RefObject := ZaberCommand);
	END_IF
END_IF
END_METHOD

METHOD set_ictrl_afcff_ss
IF ZaberStatus.ComponentStatus.iLastCommand <> 0 THEN
	ZaberStatus.ComponentStatus.iLastCommand.P_CommandStatus.LastCommandMessage := Base.F_GetLastWordInString(__POUNAME());
END_IF

IF NOT _DispatchValid() THEN
	RETURN;
ELSE
	_BuildCommandStringNoArgs();
	
	IF iBufferSend <> 0 AND __QUERYINTERFACE(iBufferSend, testIBufferSend) THEN
		iBufferSend.AddObject(RefObject := ZaberCommand);
	END_IF
END_IF
END_METHOD

METHOD set_ictrl_afcff_ss_max
IF ZaberStatus.ComponentStatus.iLastCommand <> 0 THEN
	ZaberStatus.ComponentStatus.iLastCommand.P_CommandStatus.LastCommandMessage := Base.F_GetLastWordInString(__POUNAME());
END_IF

IF NOT _DispatchValid() THEN
	RETURN;
ELSE
	_BuildCommandStringNoArgs();
	
	IF iBufferSend <> 0 AND __QUERYINTERFACE(iBufferSend, testIBufferSend) THEN
		iBufferSend.AddObject(RefObject := ZaberCommand);
	END_IF
END_IF
END_METHOD

METHOD set_ictrl_delay
IF ZaberStatus.ComponentStatus.iLastCommand <> 0 THEN
	ZaberStatus.ComponentStatus.iLastCommand.P_CommandStatus.LastCommandMessage := Base.F_GetLastWordInString(__POUNAME());
END_IF

IF NOT _DispatchValid() THEN
	RETURN;
ELSE
	_BuildCommandStringNoArgs();
	
	IF iBufferSend <> 0 AND __QUERYINTERFACE(iBufferSend, testIBufferSend) THEN
		iBufferSend.AddObject(RefObject := ZaberCommand);
	END_IF
END_IF
END_METHOD

METHOD set_ictrl_ff_kd
IF ZaberStatus.ComponentStatus.iLastCommand <> 0 THEN
	ZaberStatus.ComponentStatus.iLastCommand.P_CommandStatus.LastCommandMessage := Base.F_GetLastWordInString(__POUNAME());
END_IF

IF NOT _DispatchValid() THEN
	RETURN;
ELSE
	_BuildCommandStringNoArgs();
	
	IF iBufferSend <> 0 AND __QUERYINTERFACE(iBufferSend, testIBufferSend) THEN
		iBufferSend.AddObject(RefObject := ZaberCommand);
	END_IF
END_IF
END_METHOD

METHOD set_ictrl_ff_kp
IF ZaberStatus.ComponentStatus.iLastCommand <> 0 THEN
	ZaberStatus.ComponentStatus.iLastCommand.P_CommandStatus.LastCommandMessage := Base.F_GetLastWordInString(__POUNAME());
END_IF

IF NOT _DispatchValid() THEN
	RETURN;
ELSE
	_BuildCommandStringNoArgs();
	
	IF iBufferSend <> 0 AND __QUERYINTERFACE(iBufferSend, testIBufferSend) THEN
		iBufferSend.AddObject(RefObject := ZaberCommand);
	END_IF
END_IF
END_METHOD

METHOD set_ictrl_gain_coldmult
IF ZaberStatus.ComponentStatus.iLastCommand <> 0 THEN
	ZaberStatus.ComponentStatus.iLastCommand.P_CommandStatus.LastCommandMessage := Base.F_GetLastWordInString(__POUNAME());
END_IF

IF NOT _DispatchValid() THEN
	RETURN;
ELSE
	_BuildCommandStringNoArgs();
	
	IF iBufferSend <> 0 AND __QUERYINTERFACE(iBufferSend, testIBufferSend) THEN
		iBufferSend.AddObject(RefObject := ZaberCommand);
	END_IF
END_IF
END_METHOD

METHOD set_ictrl_period
IF ZaberStatus.ComponentStatus.iLastCommand <> 0 THEN
	ZaberStatus.ComponentStatus.iLastCommand.P_CommandStatus.LastCommandMessage := Base.F_GetLastWordInString(__POUNAME());
END_IF

IF NOT _DispatchValid() THEN
	RETURN;
ELSE
	_BuildCommandStringNoArgs();
	
	IF iBufferSend <> 0 AND __QUERYINTERFACE(iBufferSend, testIBufferSend) THEN
		iBufferSend.AddObject(RefObject := ZaberCommand);
	END_IF
END_IF
END_METHOD

METHOD set_ictrl_pi_ki
IF ZaberStatus.ComponentStatus.iLastCommand <> 0 THEN
	ZaberStatus.ComponentStatus.iLastCommand.P_CommandStatus.LastCommandMessage := Base.F_GetLastWordInString(__POUNAME());
END_IF

IF NOT _DispatchValid() THEN
	RETURN;
ELSE
	_BuildCommandStringNoArgs();
	
	IF iBufferSend <> 0 AND __QUERYINTERFACE(iBufferSend, testIBufferSend) THEN
		iBufferSend.AddObject(RefObject := ZaberCommand);
	END_IF
END_IF
END_METHOD

METHOD set_ictrl_pi_kp
IF ZaberStatus.ComponentStatus.iLastCommand <> 0 THEN
	ZaberStatus.ComponentStatus.iLastCommand.P_CommandStatus.LastCommandMessage := Base.F_GetLastWordInString(__POUNAME());
END_IF

IF NOT _DispatchValid() THEN
	RETURN;
ELSE
	_BuildCommandStringNoArgs();
	
	IF iBufferSend <> 0 AND __QUERYINTERFACE(iBufferSend, testIBufferSend) THEN
		iBufferSend.AddObject(RefObject := ZaberCommand);
	END_IF
END_IF
END_METHOD

METHOD set_ictrl_type
IF ZaberStatus.ComponentStatus.iLastCommand <> 0 THEN
	ZaberStatus.ComponentStatus.iLastCommand.P_CommandStatus.LastCommandMessage := Base.F_GetLastWordInString(__POUNAME());
END_IF

IF NOT _DispatchValid() THEN
	RETURN;
ELSE
	_BuildCommandStringNoArgs();
	
	IF iBufferSend <> 0 AND __QUERYINTERFACE(iBufferSend, testIBufferSend) THEN
		iBufferSend.AddObject(RefObject := ZaberCommand);
	END_IF
END_IF
END_METHOD

METHOD set_io_ai_1_fc
IF ZaberStatus.ComponentStatus.iLastCommand <> 0 THEN
	ZaberStatus.ComponentStatus.iLastCommand.P_CommandStatus.LastCommandMessage := Base.F_GetLastWordInString(__POUNAME());
END_IF

IF NOT _DispatchValid() THEN
	RETURN;
ELSE
	_BuildCommandStringNoArgs();
	
	IF iBufferSend <> 0 AND __QUERYINTERFACE(iBufferSend, testIBufferSend) THEN
		iBufferSend.AddObject(RefObject := ZaberCommand);
	END_IF
END_IF
END_METHOD

METHOD set_io_ai_2_fc
IF ZaberStatus.ComponentStatus.iLastCommand <> 0 THEN
	ZaberStatus.ComponentStatus.iLastCommand.P_CommandStatus.LastCommandMessage := Base.F_GetLastWordInString(__POUNAME());
END_IF

IF NOT _DispatchValid() THEN
	RETURN;
ELSE
	_BuildCommandStringNoArgs();
	
	IF iBufferSend <> 0 AND __QUERYINTERFACE(iBufferSend, testIBufferSend) THEN
		iBufferSend.AddObject(RefObject := ZaberCommand);
	END_IF
END_IF
END_METHOD

METHOD set_io_ai_3_fc
IF ZaberStatus.ComponentStatus.iLastCommand <> 0 THEN
	ZaberStatus.ComponentStatus.iLastCommand.P_CommandStatus.LastCommandMessage := Base.F_GetLastWordInString(__POUNAME());
END_IF

IF NOT _DispatchValid() THEN
	RETURN;
ELSE
	_BuildCommandStringNoArgs();
	
	IF iBufferSend <> 0 AND __QUERYINTERFACE(iBufferSend, testIBufferSend) THEN
		iBufferSend.AddObject(RefObject := ZaberCommand);
	END_IF
END_IF
END_METHOD

METHOD set_io_ai_4_fc
IF ZaberStatus.ComponentStatus.iLastCommand <> 0 THEN
	ZaberStatus.ComponentStatus.iLastCommand.P_CommandStatus.LastCommandMessage := Base.F_GetLastWordInString(__POUNAME());
END_IF

IF NOT _DispatchValid() THEN
	RETURN;
ELSE
	_BuildCommandStringNoArgs();
	
	IF iBufferSend <> 0 AND __QUERYINTERFACE(iBufferSend, testIBufferSend) THEN
		iBufferSend.AddObject(RefObject := ZaberCommand);
	END_IF
END_IF
END_METHOD

METHOD set_io_di_port
IF ZaberStatus.ComponentStatus.iLastCommand <> 0 THEN
	ZaberStatus.ComponentStatus.iLastCommand.P_CommandStatus.LastCommandMessage := Base.F_GetLastWordInString(__POUNAME());
END_IF

IF NOT _DispatchValid() THEN
	RETURN;
ELSE
	_BuildCommandStringNoArgs();
	
	IF iBufferSend <> 0 AND __QUERYINTERFACE(iBufferSend, testIBufferSend) THEN
		iBufferSend.AddObject(RefObject := ZaberCommand);
	END_IF
END_IF
END_METHOD

METHOD set_io_do_port
IF ZaberStatus.ComponentStatus.iLastCommand <> 0 THEN
	ZaberStatus.ComponentStatus.iLastCommand.P_CommandStatus.LastCommandMessage := Base.F_GetLastWordInString(__POUNAME());
END_IF

IF NOT _DispatchValid() THEN
	RETURN;
ELSE
	_BuildCommandStringNoArgs();
	
	IF iBufferSend <> 0 AND __QUERYINTERFACE(iBufferSend, testIBufferSend) THEN
		iBufferSend.AddObject(RefObject := ZaberCommand);
	END_IF
END_IF
END_METHOD

METHOD set_knob_dir
IF ZaberStatus.ComponentStatus.iLastCommand <> 0 THEN
	ZaberStatus.ComponentStatus.iLastCommand.P_CommandStatus.LastCommandMessage := Base.F_GetLastWordInString(__POUNAME());
END_IF

IF NOT _DispatchValid() THEN
	RETURN;
ELSE
	_BuildCommandStringNoArgs();
	
	IF iBufferSend <> 0 AND __QUERYINTERFACE(iBufferSend, testIBufferSend) THEN
		iBufferSend.AddObject(RefObject := ZaberCommand);
	END_IF
END_IF
END_METHOD

METHOD set_knob_distance
IF ZaberStatus.ComponentStatus.iLastCommand <> 0 THEN
	ZaberStatus.ComponentStatus.iLastCommand.P_CommandStatus.LastCommandMessage := Base.F_GetLastWordInString(__POUNAME());
END_IF

IF NOT _DispatchValid() THEN
	RETURN;
ELSE
	_BuildCommandStringNoArgs();
	
	IF iBufferSend <> 0 AND __QUERYINTERFACE(iBufferSend, testIBufferSend) THEN
		iBufferSend.AddObject(RefObject := ZaberCommand);
	END_IF
END_IF
END_METHOD

METHOD set_knob_enable
IF ZaberStatus.ComponentStatus.iLastCommand <> 0 THEN
	ZaberStatus.ComponentStatus.iLastCommand.P_CommandStatus.LastCommandMessage := Base.F_GetLastWordInString(__POUNAME());
END_IF

IF NOT _DispatchValid() THEN
	RETURN;
ELSE
	_BuildCommandStringNoArgs();
	
	IF iBufferSend <> 0 AND __QUERYINTERFACE(iBufferSend, testIBufferSend) THEN
		iBufferSend.AddObject(RefObject := ZaberCommand);
	END_IF
END_IF
END_METHOD

METHOD set_knob_maxspeed
IF ZaberStatus.ComponentStatus.iLastCommand <> 0 THEN
	ZaberStatus.ComponentStatus.iLastCommand.P_CommandStatus.LastCommandMessage := Base.F_GetLastWordInString(__POUNAME());
END_IF

IF NOT _DispatchValid() THEN
	RETURN;
ELSE
	_BuildCommandStringNoArgs();
	
	IF iBufferSend <> 0 AND __QUERYINTERFACE(iBufferSend, testIBufferSend) THEN
		iBufferSend.AddObject(RefObject := ZaberCommand);
	END_IF
END_IF
END_METHOD

METHOD set_knob_mode
IF ZaberStatus.ComponentStatus.iLastCommand <> 0 THEN
	ZaberStatus.ComponentStatus.iLastCommand.P_CommandStatus.LastCommandMessage := Base.F_GetLastWordInString(__POUNAME());
END_IF

IF NOT _DispatchValid() THEN
	RETURN;
ELSE
	_BuildCommandStringNoArgs();
	
	IF iBufferSend <> 0 AND __QUERYINTERFACE(iBufferSend, testIBufferSend) THEN
		iBufferSend.AddObject(RefObject := ZaberCommand);
	END_IF
END_IF
END_METHOD

METHOD set_knob_speedprofile
IF ZaberStatus.ComponentStatus.iLastCommand <> 0 THEN
	ZaberStatus.ComponentStatus.iLastCommand.P_CommandStatus.LastCommandMessage := Base.F_GetLastWordInString(__POUNAME());
END_IF

IF NOT _DispatchValid() THEN
	RETURN;
ELSE
	_BuildCommandStringNoArgs();
	
	IF iBufferSend <> 0 AND __QUERYINTERFACE(iBufferSend, testIBufferSend) THEN
		iBufferSend.AddObject(RefObject := ZaberCommand);
	END_IF
END_IF
END_METHOD

METHOD set_limit_approach_maxspeed
IF ZaberStatus.ComponentStatus.iLastCommand <> 0 THEN
	ZaberStatus.ComponentStatus.iLastCommand.P_CommandStatus.LastCommandMessage := Base.F_GetLastWordInString(__POUNAME());
END_IF

IF NOT _DispatchValid() THEN
	RETURN;
ELSE
	_BuildCommandStringNoArgs();
	
	IF iBufferSend <> 0 AND __QUERYINTERFACE(iBufferSend, testIBufferSend) THEN
		iBufferSend.AddObject(RefObject := ZaberCommand);
	END_IF
END_IF
END_METHOD

METHOD set_limit_detect_decelonly
IF ZaberStatus.ComponentStatus.iLastCommand <> 0 THEN
	ZaberStatus.ComponentStatus.iLastCommand.P_CommandStatus.LastCommandMessage := Base.F_GetLastWordInString(__POUNAME());
END_IF

IF NOT _DispatchValid() THEN
	RETURN;
ELSE
	_BuildCommandStringNoArgs();
	
	IF iBufferSend <> 0 AND __QUERYINTERFACE(iBufferSend, testIBufferSend) THEN
		iBufferSend.AddObject(RefObject := ZaberCommand);
	END_IF
END_IF
END_METHOD

METHOD set_limit_detect_maxspeed
IF ZaberStatus.ComponentStatus.iLastCommand <> 0 THEN
	ZaberStatus.ComponentStatus.iLastCommand.P_CommandStatus.LastCommandMessage := Base.F_GetLastWordInString(__POUNAME());
END_IF

IF NOT _DispatchValid() THEN
	RETURN;
ELSE
	_BuildCommandStringNoArgs();
	
	IF iBufferSend <> 0 AND __QUERYINTERFACE(iBufferSend, testIBufferSend) THEN
		iBufferSend.AddObject(RefObject := ZaberCommand);
	END_IF
END_IF
END_METHOD

METHOD set_limit_home_action
IF ZaberStatus.ComponentStatus.iLastCommand <> 0 THEN
	ZaberStatus.ComponentStatus.iLastCommand.P_CommandStatus.LastCommandMessage := Base.F_GetLastWordInString(__POUNAME());
END_IF

IF NOT _DispatchValid() THEN
	RETURN;
ELSE
	_BuildCommandStringNoArgs();
	
	IF iBufferSend <> 0 AND __QUERYINTERFACE(iBufferSend, testIBufferSend) THEN
		iBufferSend.AddObject(RefObject := ZaberCommand);
	END_IF
END_IF
END_METHOD

METHOD set_limit_home_bidirectional
IF ZaberStatus.ComponentStatus.iLastCommand <> 0 THEN
	ZaberStatus.ComponentStatus.iLastCommand.P_CommandStatus.LastCommandMessage := Base.F_GetLastWordInString(__POUNAME());
END_IF

IF NOT _DispatchValid() THEN
	RETURN;
ELSE
	_BuildCommandStringNoArgs();
	
	IF iBufferSend <> 0 AND __QUERYINTERFACE(iBufferSend, testIBufferSend) THEN
		iBufferSend.AddObject(RefObject := ZaberCommand);
	END_IF
END_IF
END_METHOD

METHOD set_limit_home_edge
IF ZaberStatus.ComponentStatus.iLastCommand <> 0 THEN
	ZaberStatus.ComponentStatus.iLastCommand.P_CommandStatus.LastCommandMessage := Base.F_GetLastWordInString(__POUNAME());
END_IF

IF NOT _DispatchValid() THEN
	RETURN;
ELSE
	_BuildCommandStringNoArgs();
	
	IF iBufferSend <> 0 AND __QUERYINTERFACE(iBufferSend, testIBufferSend) THEN
		iBufferSend.AddObject(RefObject := ZaberCommand);
	END_IF
END_IF
END_METHOD

METHOD set_limit_home_offset
IF ZaberStatus.ComponentStatus.iLastCommand <> 0 THEN
	ZaberStatus.ComponentStatus.iLastCommand.P_CommandStatus.LastCommandMessage := Base.F_GetLastWordInString(__POUNAME());
END_IF

IF NOT _DispatchValid() THEN
	RETURN;
ELSE
	_BuildCommandStringNoArgs();
	
	IF iBufferSend <> 0 AND __QUERYINTERFACE(iBufferSend, testIBufferSend) THEN
		iBufferSend.AddObject(RefObject := ZaberCommand);
	END_IF
END_IF
END_METHOD

METHOD set_limit_home_posupdate
IF ZaberStatus.ComponentStatus.iLastCommand <> 0 THEN
	ZaberStatus.ComponentStatus.iLastCommand.P_CommandStatus.LastCommandMessage := Base.F_GetLastWordInString(__POUNAME());
END_IF

IF NOT _DispatchValid() THEN
	RETURN;
ELSE
	_BuildCommandStringNoArgs();
	
	IF iBufferSend <> 0 AND __QUERYINTERFACE(iBufferSend, testIBufferSend) THEN
		iBufferSend.AddObject(RefObject := ZaberCommand);
	END_IF
END_IF
END_METHOD

METHOD set_limit_home_preset
IF ZaberStatus.ComponentStatus.iLastCommand <> 0 THEN
	ZaberStatus.ComponentStatus.iLastCommand.P_CommandStatus.LastCommandMessage := Base.F_GetLastWordInString(__POUNAME());
END_IF

IF NOT _DispatchValid() THEN
	RETURN;
ELSE
	_BuildCommandStringNoArgs();
	
	IF iBufferSend <> 0 AND __QUERYINTERFACE(iBufferSend, testIBufferSend) THEN
		iBufferSend.AddObject(RefObject := ZaberCommand);
	END_IF
END_IF
END_METHOD

METHOD set_limit_home_source
IF ZaberStatus.ComponentStatus.iLastCommand <> 0 THEN
	ZaberStatus.ComponentStatus.iLastCommand.P_CommandStatus.LastCommandMessage := Base.F_GetLastWordInString(__POUNAME());
END_IF

IF NOT _DispatchValid() THEN
	RETURN;
ELSE
	_BuildCommandStringNoArgs();
	
	IF iBufferSend <> 0 AND __QUERYINTERFACE(iBufferSend, testIBufferSend) THEN
		iBufferSend.AddObject(RefObject := ZaberCommand);
	END_IF
END_IF
END_METHOD

METHOD set_limit_home_state
IF ZaberStatus.ComponentStatus.iLastCommand <> 0 THEN
	ZaberStatus.ComponentStatus.iLastCommand.P_CommandStatus.LastCommandMessage := Base.F_GetLastWordInString(__POUNAME());
END_IF

IF NOT _DispatchValid() THEN
	RETURN;
ELSE
	_BuildCommandStringNoArgs();
	
	IF iBufferSend <> 0 AND __QUERYINTERFACE(iBufferSend, testIBufferSend) THEN
		iBufferSend.AddObject(RefObject := ZaberCommand);
	END_IF
END_IF
END_METHOD

METHOD set_limit_home_triggered
IF ZaberStatus.ComponentStatus.iLastCommand <> 0 THEN
	ZaberStatus.ComponentStatus.iLastCommand.P_CommandStatus.LastCommandMessage := Base.F_GetLastWordInString(__POUNAME());
END_IF

IF NOT _DispatchValid() THEN
	RETURN;
ELSE
	_BuildCommandStringNoArgs();
	
	IF iBufferSend <> 0 AND __QUERYINTERFACE(iBufferSend, testIBufferSend) THEN
		iBufferSend.AddObject(RefObject := ZaberCommand);
	END_IF
END_IF
END_METHOD

METHOD set_limit_home_tune
IF ZaberStatus.ComponentStatus.iLastCommand <> 0 THEN
	ZaberStatus.ComponentStatus.iLastCommand.P_CommandStatus.LastCommandMessage := Base.F_GetLastWordInString(__POUNAME());
END_IF

IF NOT _DispatchValid() THEN
	RETURN;
ELSE
	_BuildCommandStringNoArgs();
	
	IF iBufferSend <> 0 AND __QUERYINTERFACE(iBufferSend, testIBufferSend) THEN
		iBufferSend.AddObject(RefObject := ZaberCommand);
	END_IF
END_IF
END_METHOD

METHOD set_limit_home_type
IF ZaberStatus.ComponentStatus.iLastCommand <> 0 THEN
	ZaberStatus.ComponentStatus.iLastCommand.P_CommandStatus.LastCommandMessage := Base.F_GetLastWordInString(__POUNAME());
END_IF

IF NOT _DispatchValid() THEN
	RETURN;
ELSE
	_BuildCommandStringNoArgs();
	
	IF iBufferSend <> 0 AND __QUERYINTERFACE(iBufferSend, testIBufferSend) THEN
		iBufferSend.AddObject(RefObject := ZaberCommand);
	END_IF
END_IF
END_METHOD

METHOD set_limit_home_width
IF ZaberStatus.ComponentStatus.iLastCommand <> 0 THEN
	ZaberStatus.ComponentStatus.iLastCommand.P_CommandStatus.LastCommandMessage := Base.F_GetLastWordInString(__POUNAME());
END_IF

IF NOT _DispatchValid() THEN
	RETURN;
ELSE
	_BuildCommandStringNoArgs();
	
	IF iBufferSend <> 0 AND __QUERYINTERFACE(iBufferSend, testIBufferSend) THEN
		iBufferSend.AddObject(RefObject := ZaberCommand);
	END_IF
END_IF
END_METHOD

METHOD set_limit_max
IF ZaberStatus.ComponentStatus.iLastCommand <> 0 THEN
	ZaberStatus.ComponentStatus.iLastCommand.P_CommandStatus.LastCommandMessage := Base.F_GetLastWordInString(__POUNAME());
END_IF

IF NOT _DispatchValid() THEN
	RETURN;
ELSE
	_BuildCommandStringNoArgs();
	
	IF iBufferSend <> 0 AND __QUERYINTERFACE(iBufferSend, testIBufferSend) THEN
		iBufferSend.AddObject(RefObject := ZaberCommand);
	END_IF
END_IF
END_METHOD

METHOD set_limit_min
IF ZaberStatus.ComponentStatus.iLastCommand <> 0 THEN
	ZaberStatus.ComponentStatus.iLastCommand.P_CommandStatus.LastCommandMessage := Base.F_GetLastWordInString(__POUNAME());
END_IF

IF NOT _DispatchValid() THEN
	RETURN;
ELSE
	_BuildCommandStringNoArgs();
	
	IF iBufferSend <> 0 AND __QUERYINTERFACE(iBufferSend, testIBufferSend) THEN
		iBufferSend.AddObject(RefObject := ZaberCommand);
	END_IF
END_IF
END_METHOD

METHOD set_limit_range_mode
IF ZaberStatus.ComponentStatus.iLastCommand <> 0 THEN
	ZaberStatus.ComponentStatus.iLastCommand.P_CommandStatus.LastCommandMessage := Base.F_GetLastWordInString(__POUNAME());
END_IF

IF NOT _DispatchValid() THEN
	RETURN;
ELSE
	_BuildCommandStringNoArgs();
	
	IF iBufferSend <> 0 AND __QUERYINTERFACE(iBufferSend, testIBufferSend) THEN
		iBufferSend.AddObject(RefObject := ZaberCommand);
	END_IF
END_IF
END_METHOD

METHOD set_lockstep_numgroups
IF ZaberStatus.ComponentStatus.iLastCommand <> 0 THEN
	ZaberStatus.ComponentStatus.iLastCommand.P_CommandStatus.LastCommandMessage := Base.F_GetLastWordInString(__POUNAME());
END_IF

IF NOT _DispatchValid() THEN
	RETURN;
ELSE
	_BuildCommandStringNoArgs();
	
	IF iBufferSend <> 0 AND __QUERYINTERFACE(iBufferSend, testIBufferSend) THEN
		iBufferSend.AddObject(RefObject := ZaberCommand);
	END_IF
END_IF
END_METHOD

METHOD set_maxspeed
IF ZaberStatus.ComponentStatus.iLastCommand <> 0 THEN
	ZaberStatus.ComponentStatus.iLastCommand.P_CommandStatus.LastCommandMessage := Base.F_GetLastWordInString(__POUNAME());
END_IF

IF NOT _DispatchValid() THEN
	RETURN;
ELSE
	_BuildCommandStringNoArgs();
	
	IF iBufferSend <> 0 AND __QUERYINTERFACE(iBufferSend, testIBufferSend) THEN
		iBufferSend.AddObject(RefObject := ZaberCommand);
	END_IF
END_IF
END_METHOD

METHOD set_motion_accel_ramptime
IF ZaberStatus.ComponentStatus.iLastCommand <> 0 THEN
	ZaberStatus.ComponentStatus.iLastCommand.P_CommandStatus.LastCommandMessage := Base.F_GetLastWordInString(__POUNAME());
END_IF

IF NOT _DispatchValid() THEN
	RETURN;
ELSE
	_BuildCommandStringNoArgs();
	
	IF iBufferSend <> 0 AND __QUERYINTERFACE(iBufferSend, testIBufferSend) THEN
		iBufferSend.AddObject(RefObject := ZaberCommand);
	END_IF
END_IF
END_METHOD

METHOD set_motion_accelonly
IF ZaberStatus.ComponentStatus.iLastCommand <> 0 THEN
	ZaberStatus.ComponentStatus.iLastCommand.P_CommandStatus.LastCommandMessage := Base.F_GetLastWordInString(__POUNAME());
END_IF

IF NOT _DispatchValid() THEN
	RETURN;
ELSE
	_BuildCommandStringNoArgs();
	
	IF iBufferSend <> 0 AND __QUERYINTERFACE(iBufferSend, testIBufferSend) THEN
		iBufferSend.AddObject(RefObject := ZaberCommand);
	END_IF
END_IF
END_METHOD

METHOD set_motion_busy
IF ZaberStatus.ComponentStatus.iLastCommand <> 0 THEN
	ZaberStatus.ComponentStatus.iLastCommand.P_CommandStatus.LastCommandMessage := Base.F_GetLastWordInString(__POUNAME());
END_IF

IF NOT _DispatchValid() THEN
	RETURN;
ELSE
	_BuildCommandStringNoArgs();
	
	IF iBufferSend <> 0 AND __QUERYINTERFACE(iBufferSend, testIBufferSend) THEN
		iBufferSend.AddObject(RefObject := ZaberCommand);
	END_IF
END_IF
END_METHOD

METHOD set_motion_decelonly
IF ZaberStatus.ComponentStatus.iLastCommand <> 0 THEN
	ZaberStatus.ComponentStatus.iLastCommand.P_CommandStatus.LastCommandMessage := Base.F_GetLastWordInString(__POUNAME());
END_IF

IF NOT _DispatchValid() THEN
	RETURN;
ELSE
	_BuildCommandStringNoArgs();
	
	IF iBufferSend <> 0 AND __QUERYINTERFACE(iBufferSend, testIBufferSend) THEN
		iBufferSend.AddObject(RefObject := ZaberCommand);
	END_IF
END_IF
END_METHOD

METHOD set_motion_index_dist
IF ZaberStatus.ComponentStatus.iLastCommand <> 0 THEN
	ZaberStatus.ComponentStatus.iLastCommand.P_CommandStatus.LastCommandMessage := Base.F_GetLastWordInString(__POUNAME());
END_IF

IF NOT _DispatchValid() THEN
	RETURN;
ELSE
	_BuildCommandStringNoArgs();
	
	IF iBufferSend <> 0 AND __QUERYINTERFACE(iBufferSend, testIBufferSend) THEN
		iBufferSend.AddObject(RefObject := ZaberCommand);
	END_IF
END_IF
END_METHOD

METHOD set_motion_index_num
IF ZaberStatus.ComponentStatus.iLastCommand <> 0 THEN
	ZaberStatus.ComponentStatus.iLastCommand.P_CommandStatus.LastCommandMessage := Base.F_GetLastWordInString(__POUNAME());
END_IF

IF NOT _DispatchValid() THEN
	RETURN;
ELSE
	_BuildCommandStringNoArgs();
	
	IF iBufferSend <> 0 AND __QUERYINTERFACE(iBufferSend, testIBufferSend) THEN
		iBufferSend.AddObject(RefObject := ZaberCommand);
	END_IF
END_IF
END_METHOD

METHOD set_motion_tracking_ai
IF ZaberStatus.ComponentStatus.iLastCommand <> 0 THEN
	ZaberStatus.ComponentStatus.iLastCommand.P_CommandStatus.LastCommandMessage := Base.F_GetLastWordInString(__POUNAME());
END_IF

IF NOT _DispatchValid() THEN
	RETURN;
ELSE
	_BuildCommandStringNoArgs();
	
	IF iBufferSend <> 0 AND __QUERYINTERFACE(iBufferSend, testIBufferSend) THEN
		iBufferSend.AddObject(RefObject := ZaberCommand);
	END_IF
END_IF
END_METHOD

METHOD set_motion_tracking_dir
IF ZaberStatus.ComponentStatus.iLastCommand <> 0 THEN
	ZaberStatus.ComponentStatus.iLastCommand.P_CommandStatus.LastCommandMessage := Base.F_GetLastWordInString(__POUNAME());
END_IF

IF NOT _DispatchValid() THEN
	RETURN;
ELSE
	_BuildCommandStringNoArgs();
	
	IF iBufferSend <> 0 AND __QUERYINTERFACE(iBufferSend, testIBufferSend) THEN
		iBufferSend.AddObject(RefObject := ZaberCommand);
	END_IF
END_IF
END_METHOD

METHOD set_motion_tracking_ki
IF ZaberStatus.ComponentStatus.iLastCommand <> 0 THEN
	ZaberStatus.ComponentStatus.iLastCommand.P_CommandStatus.LastCommandMessage := Base.F_GetLastWordInString(__POUNAME());
END_IF

IF NOT _DispatchValid() THEN
	RETURN;
ELSE
	_BuildCommandStringNoArgs();
	
	IF iBufferSend <> 0 AND __QUERYINTERFACE(iBufferSend, testIBufferSend) THEN
		iBufferSend.AddObject(RefObject := ZaberCommand);
	END_IF
END_IF
END_METHOD

METHOD set_motion_tracking_kp
IF ZaberStatus.ComponentStatus.iLastCommand <> 0 THEN
	ZaberStatus.ComponentStatus.iLastCommand.P_CommandStatus.LastCommandMessage := Base.F_GetLastWordInString(__POUNAME());
END_IF

IF NOT _DispatchValid() THEN
	RETURN;
ELSE
	_BuildCommandStringNoArgs();
	
	IF iBufferSend <> 0 AND __QUERYINTERFACE(iBufferSend, testIBufferSend) THEN
		iBufferSend.AddObject(RefObject := ZaberCommand);
	END_IF
END_IF
END_METHOD

METHOD set_motion_tracking_limit_max
IF ZaberStatus.ComponentStatus.iLastCommand <> 0 THEN
	ZaberStatus.ComponentStatus.iLastCommand.P_CommandStatus.LastCommandMessage := Base.F_GetLastWordInString(__POUNAME());
END_IF

IF NOT _DispatchValid() THEN
	RETURN;
ELSE
	_BuildCommandStringNoArgs();
	
	IF iBufferSend <> 0 AND __QUERYINTERFACE(iBufferSend, testIBufferSend) THEN
		iBufferSend.AddObject(RefObject := ZaberCommand);
	END_IF
END_IF
END_METHOD

METHOD set_motion_tracking_limit_min
IF ZaberStatus.ComponentStatus.iLastCommand <> 0 THEN
	ZaberStatus.ComponentStatus.iLastCommand.P_CommandStatus.LastCommandMessage := Base.F_GetLastWordInString(__POUNAME());
END_IF

IF NOT _DispatchValid() THEN
	RETURN;
ELSE
	_BuildCommandStringNoArgs();
	
	IF iBufferSend <> 0 AND __QUERYINTERFACE(iBufferSend, testIBufferSend) THEN
		iBufferSend.AddObject(RefObject := ZaberCommand);
	END_IF
END_IF
END_METHOD

METHOD set_motion_tracking_scan_dir
IF ZaberStatus.ComponentStatus.iLastCommand <> 0 THEN
	ZaberStatus.ComponentStatus.iLastCommand.P_CommandStatus.LastCommandMessage := Base.F_GetLastWordInString(__POUNAME());
END_IF

IF NOT _DispatchValid() THEN
	RETURN;
ELSE
	_BuildCommandStringNoArgs();
	
	IF iBufferSend <> 0 AND __QUERYINTERFACE(iBufferSend, testIBufferSend) THEN
		iBufferSend.AddObject(RefObject := ZaberCommand);
	END_IF
END_IF
END_METHOD

METHOD set_motion_tracking_scan_maxspeed
IF ZaberStatus.ComponentStatus.iLastCommand <> 0 THEN
	ZaberStatus.ComponentStatus.iLastCommand.P_CommandStatus.LastCommandMessage := Base.F_GetLastWordInString(__POUNAME());
END_IF

IF NOT _DispatchValid() THEN
	RETURN;
ELSE
	_BuildCommandStringNoArgs();
	
	IF iBufferSend <> 0 AND __QUERYINTERFACE(iBufferSend, testIBufferSend) THEN
		iBufferSend.AddObject(RefObject := ZaberCommand);
	END_IF
END_IF
END_METHOD

METHOD set_motion_tracking_scan_offset
IF ZaberStatus.ComponentStatus.iLastCommand <> 0 THEN
	ZaberStatus.ComponentStatus.iLastCommand.P_CommandStatus.LastCommandMessage := Base.F_GetLastWordInString(__POUNAME());
END_IF

IF NOT _DispatchValid() THEN
	RETURN;
ELSE
	_BuildCommandStringNoArgs();
	
	IF iBufferSend <> 0 AND __QUERYINTERFACE(iBufferSend, testIBufferSend) THEN
		iBufferSend.AddObject(RefObject := ZaberCommand);
	END_IF
END_IF
END_METHOD

METHOD set_motion_tracking_scan_period
IF ZaberStatus.ComponentStatus.iLastCommand <> 0 THEN
	ZaberStatus.ComponentStatus.iLastCommand.P_CommandStatus.LastCommandMessage := Base.F_GetLastWordInString(__POUNAME());
END_IF

IF NOT _DispatchValid() THEN
	RETURN;
ELSE
	_BuildCommandStringNoArgs();
	
	IF iBufferSend <> 0 AND __QUERYINTERFACE(iBufferSend, testIBufferSend) THEN
		iBufferSend.AddObject(RefObject := ZaberCommand);
	END_IF
END_IF
END_METHOD

METHOD set_motion_tracking_scan_signal_valid_delay
IF ZaberStatus.ComponentStatus.iLastCommand <> 0 THEN
	ZaberStatus.ComponentStatus.iLastCommand.P_CommandStatus.LastCommandMessage := Base.F_GetLastWordInString(__POUNAME());
END_IF

IF NOT _DispatchValid() THEN
	RETURN;
ELSE
	_BuildCommandStringNoArgs();
	
	IF iBufferSend <> 0 AND __QUERYINTERFACE(iBufferSend, testIBufferSend) THEN
		iBufferSend.AddObject(RefObject := ZaberCommand);
	END_IF
END_IF
END_METHOD

METHOD set_motion_tracking_scan_tolerance
IF ZaberStatus.ComponentStatus.iLastCommand <> 0 THEN
	ZaberStatus.ComponentStatus.iLastCommand.P_CommandStatus.LastCommandMessage := Base.F_GetLastWordInString(__POUNAME());
END_IF

IF NOT _DispatchValid() THEN
	RETURN;
ELSE
	_BuildCommandStringNoArgs();
	
	IF iBufferSend <> 0 AND __QUERYINTERFACE(iBufferSend, testIBufferSend) THEN
		iBufferSend.AddObject(RefObject := ZaberCommand);
	END_IF
END_IF
END_METHOD

METHOD set_motion_tracking_setpoint
IF ZaberStatus.ComponentStatus.iLastCommand <> 0 THEN
	ZaberStatus.ComponentStatus.iLastCommand.P_CommandStatus.LastCommandMessage := Base.F_GetLastWordInString(__POUNAME());
END_IF

IF NOT _DispatchValid() THEN
	RETURN;
ELSE
	_BuildCommandStringNoArgs();
	
	IF iBufferSend <> 0 AND __QUERYINTERFACE(iBufferSend, testIBufferSend) THEN
		iBufferSend.AddObject(RefObject := ZaberCommand);
	END_IF
END_IF
END_METHOD

METHOD set_motion_tracking_settle_period
IF ZaberStatus.ComponentStatus.iLastCommand <> 0 THEN
	ZaberStatus.ComponentStatus.iLastCommand.P_CommandStatus.LastCommandMessage := Base.F_GetLastWordInString(__POUNAME());
END_IF

IF NOT _DispatchValid() THEN
	RETURN;
ELSE
	_BuildCommandStringNoArgs();
	
	IF iBufferSend <> 0 AND __QUERYINTERFACE(iBufferSend, testIBufferSend) THEN
		iBufferSend.AddObject(RefObject := ZaberCommand);
	END_IF
END_IF
END_METHOD

METHOD set_motion_tracking_settle_tolerance
IF ZaberStatus.ComponentStatus.iLastCommand <> 0 THEN
	ZaberStatus.ComponentStatus.iLastCommand.P_CommandStatus.LastCommandMessage := Base.F_GetLastWordInString(__POUNAME());
END_IF

IF NOT _DispatchValid() THEN
	RETURN;
ELSE
	_BuildCommandStringNoArgs();
	
	IF iBufferSend <> 0 AND __QUERYINTERFACE(iBufferSend, testIBufferSend) THEN
		iBufferSend.AddObject(RefObject := ZaberCommand);
	END_IF
END_IF
END_METHOD

METHOD set_motion_tracking_settle_tolerance_met
IF ZaberStatus.ComponentStatus.iLastCommand <> 0 THEN
	ZaberStatus.ComponentStatus.iLastCommand.P_CommandStatus.LastCommandMessage := Base.F_GetLastWordInString(__POUNAME());
END_IF

IF NOT _DispatchValid() THEN
	RETURN;
ELSE
	_BuildCommandStringNoArgs();
	
	IF iBufferSend <> 0 AND __QUERYINTERFACE(iBufferSend, testIBufferSend) THEN
		iBufferSend.AddObject(RefObject := ZaberCommand);
	END_IF
END_IF
END_METHOD

METHOD set_motion_tracking_settled
IF ZaberStatus.ComponentStatus.iLastCommand <> 0 THEN
	ZaberStatus.ComponentStatus.iLastCommand.P_CommandStatus.LastCommandMessage := Base.F_GetLastWordInString(__POUNAME());
END_IF

IF NOT _DispatchValid() THEN
	RETURN;
ELSE
	_BuildCommandStringNoArgs();
	
	IF iBufferSend <> 0 AND __QUERYINTERFACE(iBufferSend, testIBufferSend) THEN
		iBufferSend.AddObject(RefObject := ZaberCommand);
	END_IF
END_IF
END_METHOD

METHOD set_motion_tracking_signal_valid_di
IF ZaberStatus.ComponentStatus.iLastCommand <> 0 THEN
	ZaberStatus.ComponentStatus.iLastCommand.P_CommandStatus.LastCommandMessage := Base.F_GetLastWordInString(__POUNAME());
END_IF

IF NOT _DispatchValid() THEN
	RETURN;
ELSE
	_BuildCommandStringNoArgs();
	
	IF iBufferSend <> 0 AND __QUERYINTERFACE(iBufferSend, testIBufferSend) THEN
		iBufferSend.AddObject(RefObject := ZaberCommand);
	END_IF
END_IF
END_METHOD

METHOD set_motor_current_max
IF ZaberStatus.ComponentStatus.iLastCommand <> 0 THEN
	ZaberStatus.ComponentStatus.iLastCommand.P_CommandStatus.LastCommandMessage := Base.F_GetLastWordInString(__POUNAME());
END_IF

IF NOT _DispatchValid() THEN
	RETURN;
ELSE
	_BuildCommandStringNoArgs();
	
	IF iBufferSend <> 0 AND __QUERYINTERFACE(iBufferSend, testIBufferSend) THEN
		iBufferSend.AddObject(RefObject := ZaberCommand);
	END_IF
END_IF
END_METHOD

METHOD set_motor_inductance
IF ZaberStatus.ComponentStatus.iLastCommand <> 0 THEN
	ZaberStatus.ComponentStatus.iLastCommand.P_CommandStatus.LastCommandMessage := Base.F_GetLastWordInString(__POUNAME());
END_IF

IF NOT _DispatchValid() THEN
	RETURN;
ELSE
	_BuildCommandStringNoArgs();
	
	IF iBufferSend <> 0 AND __QUERYINTERFACE(iBufferSend, testIBufferSend) THEN
		iBufferSend.AddObject(RefObject := ZaberCommand);
	END_IF
END_IF
END_METHOD

METHOD set_motor_ke
IF ZaberStatus.ComponentStatus.iLastCommand <> 0 THEN
	ZaberStatus.ComponentStatus.iLastCommand.P_CommandStatus.LastCommandMessage := Base.F_GetLastWordInString(__POUNAME());
END_IF

IF NOT _DispatchValid() THEN
	RETURN;
ELSE
	_BuildCommandStringNoArgs();
	
	IF iBufferSend <> 0 AND __QUERYINTERFACE(iBufferSend, testIBufferSend) THEN
		iBufferSend.AddObject(RefObject := ZaberCommand);
	END_IF
END_IF
END_METHOD

METHOD set_motor_phase
IF ZaberStatus.ComponentStatus.iLastCommand <> 0 THEN
	ZaberStatus.ComponentStatus.iLastCommand.P_CommandStatus.LastCommandMessage := Base.F_GetLastWordInString(__POUNAME());
END_IF

IF NOT _DispatchValid() THEN
	RETURN;
ELSE
	_BuildCommandStringNoArgs();
	
	IF iBufferSend <> 0 AND __QUERYINTERFACE(iBufferSend, testIBufferSend) THEN
		iBufferSend.AddObject(RefObject := ZaberCommand);
	END_IF
END_IF
END_METHOD

METHOD set_motor_phase_ratio_div1
IF ZaberStatus.ComponentStatus.iLastCommand <> 0 THEN
	ZaberStatus.ComponentStatus.iLastCommand.P_CommandStatus.LastCommandMessage := Base.F_GetLastWordInString(__POUNAME());
END_IF

IF NOT _DispatchValid() THEN
	RETURN;
ELSE
	_BuildCommandStringNoArgs();
	
	IF iBufferSend <> 0 AND __QUERYINTERFACE(iBufferSend, testIBufferSend) THEN
		iBufferSend.AddObject(RefObject := ZaberCommand);
	END_IF
END_IF
END_METHOD

METHOD set_motor_phase_ratio_div2
IF ZaberStatus.ComponentStatus.iLastCommand <> 0 THEN
	ZaberStatus.ComponentStatus.iLastCommand.P_CommandStatus.LastCommandMessage := Base.F_GetLastWordInString(__POUNAME());
END_IF

IF NOT _DispatchValid() THEN
	RETURN;
ELSE
	_BuildCommandStringNoArgs();
	
	IF iBufferSend <> 0 AND __QUERYINTERFACE(iBufferSend, testIBufferSend) THEN
		iBufferSend.AddObject(RefObject := ZaberCommand);
	END_IF
END_IF
END_METHOD

METHOD set_motor_phase_ratio_mult
IF ZaberStatus.ComponentStatus.iLastCommand <> 0 THEN
	ZaberStatus.ComponentStatus.iLastCommand.P_CommandStatus.LastCommandMessage := Base.F_GetLastWordInString(__POUNAME());
END_IF

IF NOT _DispatchValid() THEN
	RETURN;
ELSE
	_BuildCommandStringNoArgs();
	
	IF iBufferSend <> 0 AND __QUERYINTERFACE(iBufferSend, testIBufferSend) THEN
		iBufferSend.AddObject(RefObject := ZaberCommand);
	END_IF
END_IF
END_METHOD

METHOD set_motor_resistance
IF ZaberStatus.ComponentStatus.iLastCommand <> 0 THEN
	ZaberStatus.ComponentStatus.iLastCommand.P_CommandStatus.LastCommandMessage := Base.F_GetLastWordInString(__POUNAME());
END_IF

IF NOT _DispatchValid() THEN
	RETURN;
ELSE
	_BuildCommandStringNoArgs();
	
	IF iBufferSend <> 0 AND __QUERYINTERFACE(iBufferSend, testIBufferSend) THEN
		iBufferSend.AddObject(RefObject := ZaberCommand);
	END_IF
END_IF
END_METHOD

METHOD set_parking_state
IF ZaberStatus.ComponentStatus.iLastCommand <> 0 THEN
	ZaberStatus.ComponentStatus.iLastCommand.P_CommandStatus.LastCommandMessage := Base.F_GetLastWordInString(__POUNAME());
END_IF

IF NOT _DispatchValid() THEN
	RETURN;
ELSE
	_BuildCommandStringNoArgs();
	
	IF iBufferSend <> 0 AND __QUERYINTERFACE(iBufferSend, testIBufferSend) THEN
		iBufferSend.AddObject(RefObject := ZaberCommand);
	END_IF
END_IF
END_METHOD

METHOD set_peripheral_hw_modified
IF ZaberStatus.ComponentStatus.iLastCommand <> 0 THEN
	ZaberStatus.ComponentStatus.iLastCommand.P_CommandStatus.LastCommandMessage := Base.F_GetLastWordInString(__POUNAME());
END_IF

IF NOT _DispatchValid() THEN
	RETURN;
ELSE
	_BuildCommandStringNoArgs();
	
	IF iBufferSend <> 0 AND __QUERYINTERFACE(iBufferSend, testIBufferSend) THEN
		iBufferSend.AddObject(RefObject := ZaberCommand);
	END_IF
END_IF
END_METHOD

METHOD set_peripheral_id
IF ZaberStatus.ComponentStatus.iLastCommand <> 0 THEN
	ZaberStatus.ComponentStatus.iLastCommand.P_CommandStatus.LastCommandMessage := Base.F_GetLastWordInString(__POUNAME());
END_IF

IF NOT _DispatchValid() THEN
	RETURN;
ELSE
	_BuildCommandStringNoArgs();
	
	IF iBufferSend <> 0 AND __QUERYINTERFACE(iBufferSend, testIBufferSend) THEN
		iBufferSend.AddObject(RefObject := ZaberCommand);
	END_IF
END_IF
END_METHOD

METHOD set_peripheral_id_pending
IF ZaberStatus.ComponentStatus.iLastCommand <> 0 THEN
	ZaberStatus.ComponentStatus.iLastCommand.P_CommandStatus.LastCommandMessage := Base.F_GetLastWordInString(__POUNAME());
END_IF

IF NOT _DispatchValid() THEN
	RETURN;
ELSE
	_BuildCommandStringNoArgs();
	
	IF iBufferSend <> 0 AND __QUERYINTERFACE(iBufferSend, testIBufferSend) THEN
		iBufferSend.AddObject(RefObject := ZaberCommand);
	END_IF
END_IF
END_METHOD

METHOD set_peripheral_serial
IF ZaberStatus.ComponentStatus.iLastCommand <> 0 THEN
	ZaberStatus.ComponentStatus.iLastCommand.P_CommandStatus.LastCommandMessage := Base.F_GetLastWordInString(__POUNAME());
END_IF

IF NOT _DispatchValid() THEN
	RETURN;
ELSE
	_BuildCommandStringNoArgs();
	
	IF iBufferSend <> 0 AND __QUERYINTERFACE(iBufferSend, testIBufferSend) THEN
		iBufferSend.AddObject(RefObject := ZaberCommand);
	END_IF
END_IF
END_METHOD

METHOD set_peripheral_serial_pending
IF ZaberStatus.ComponentStatus.iLastCommand <> 0 THEN
	ZaberStatus.ComponentStatus.iLastCommand.P_CommandStatus.LastCommandMessage := Base.F_GetLastWordInString(__POUNAME());
END_IF

IF NOT _DispatchValid() THEN
	RETURN;
ELSE
	_BuildCommandStringNoArgs();
	
	IF iBufferSend <> 0 AND __QUERYINTERFACE(iBufferSend, testIBufferSend) THEN
		iBufferSend.AddObject(RefObject := ZaberCommand);
	END_IF
END_IF
END_METHOD

METHOD set_pos
IF ZaberStatus.ComponentStatus.iLastCommand <> 0 THEN
	ZaberStatus.ComponentStatus.iLastCommand.P_CommandStatus.LastCommandMessage := Base.F_GetLastWordInString(__POUNAME());
END_IF

IF NOT _DispatchValid() THEN
	RETURN;
ELSE
	_BuildCommandStringNoArgs();
	
	IF iBufferSend <> 0 AND __QUERYINTERFACE(iBufferSend, testIBufferSend) THEN
		iBufferSend.AddObject(RefObject := ZaberCommand);
	END_IF
END_IF
END_METHOD

METHOD set_pvt_numseqs
IF ZaberStatus.ComponentStatus.iLastCommand <> 0 THEN
	ZaberStatus.ComponentStatus.iLastCommand.P_CommandStatus.LastCommandMessage := Base.F_GetLastWordInString(__POUNAME());
END_IF

IF NOT _DispatchValid() THEN
	RETURN;
ELSE
	_BuildCommandStringNoArgs();
	
	IF iBufferSend <> 0 AND __QUERYINTERFACE(iBufferSend, testIBufferSend) THEN
		iBufferSend.AddObject(RefObject := ZaberCommand);
	END_IF
END_IF
END_METHOD

METHOD set_resolution
IF ZaberStatus.ComponentStatus.iLastCommand <> 0 THEN
	ZaberStatus.ComponentStatus.iLastCommand.P_CommandStatus.LastCommandMessage := Base.F_GetLastWordInString(__POUNAME());
END_IF

IF NOT _DispatchValid() THEN
	RETURN;
ELSE
	_BuildCommandStringNoArgs();
	
	IF iBufferSend <> 0 AND __QUERYINTERFACE(iBufferSend, testIBufferSend) THEN
		iBufferSend.AddObject(RefObject := ZaberCommand);
	END_IF
END_IF
END_METHOD

METHOD set_scope_channel_size
IF ZaberStatus.ComponentStatus.iLastCommand <> 0 THEN
	ZaberStatus.ComponentStatus.iLastCommand.P_CommandStatus.LastCommandMessage := Base.F_GetLastWordInString(__POUNAME());
END_IF

IF NOT _DispatchValid() THEN
	RETURN;
ELSE
	_BuildCommandStringNoArgs();
	
	IF iBufferSend <> 0 AND __QUERYINTERFACE(iBufferSend, testIBufferSend) THEN
		iBufferSend.AddObject(RefObject := ZaberCommand);
	END_IF
END_IF
END_METHOD

METHOD set_scope_channel_size_max
IF ZaberStatus.ComponentStatus.iLastCommand <> 0 THEN
	ZaberStatus.ComponentStatus.iLastCommand.P_CommandStatus.LastCommandMessage := Base.F_GetLastWordInString(__POUNAME());
END_IF

IF NOT _DispatchValid() THEN
	RETURN;
ELSE
	_BuildCommandStringNoArgs();
	
	IF iBufferSend <> 0 AND __QUERYINTERFACE(iBufferSend, testIBufferSend) THEN
		iBufferSend.AddObject(RefObject := ZaberCommand);
	END_IF
END_IF
END_METHOD

METHOD set_scope_delay
IF ZaberStatus.ComponentStatus.iLastCommand <> 0 THEN
	ZaberStatus.ComponentStatus.iLastCommand.P_CommandStatus.LastCommandMessage := Base.F_GetLastWordInString(__POUNAME());
END_IF

IF NOT _DispatchValid() THEN
	RETURN;
ELSE
	_BuildCommandStringNoArgs();
	
	IF iBufferSend <> 0 AND __QUERYINTERFACE(iBufferSend, testIBufferSend) THEN
		iBufferSend.AddObject(RefObject := ZaberCommand);
	END_IF
END_IF
END_METHOD

METHOD set_scope_numchannels
IF ZaberStatus.ComponentStatus.iLastCommand <> 0 THEN
	ZaberStatus.ComponentStatus.iLastCommand.P_CommandStatus.LastCommandMessage := Base.F_GetLastWordInString(__POUNAME());
END_IF

IF NOT _DispatchValid() THEN
	RETURN;
ELSE
	_BuildCommandStringNoArgs();
	
	IF iBufferSend <> 0 AND __QUERYINTERFACE(iBufferSend, testIBufferSend) THEN
		iBufferSend.AddObject(RefObject := ZaberCommand);
	END_IF
END_IF
END_METHOD

METHOD set_scope_timebase
IF ZaberStatus.ComponentStatus.iLastCommand <> 0 THEN
	ZaberStatus.ComponentStatus.iLastCommand.P_CommandStatus.LastCommandMessage := Base.F_GetLastWordInString(__POUNAME());
END_IF

IF NOT _DispatchValid() THEN
	RETURN;
ELSE
	_BuildCommandStringNoArgs();
	
	IF iBufferSend <> 0 AND __QUERYINTERFACE(iBufferSend, testIBufferSend) THEN
		iBufferSend.AddObject(RefObject := ZaberCommand);
	END_IF
END_IF
END_METHOD

METHOD set_stream_numbufs
IF ZaberStatus.ComponentStatus.iLastCommand <> 0 THEN
	ZaberStatus.ComponentStatus.iLastCommand.P_CommandStatus.LastCommandMessage := Base.F_GetLastWordInString(__POUNAME());
END_IF

IF NOT _DispatchValid() THEN
	RETURN;
ELSE
	_BuildCommandStringNoArgs();
	
	IF iBufferSend <> 0 AND __QUERYINTERFACE(iBufferSend, testIBufferSend) THEN
		iBufferSend.AddObject(RefObject := ZaberCommand);
	END_IF
END_IF
END_METHOD

METHOD set_stream_numstreams
IF ZaberStatus.ComponentStatus.iLastCommand <> 0 THEN
	ZaberStatus.ComponentStatus.iLastCommand.P_CommandStatus.LastCommandMessage := Base.F_GetLastWordInString(__POUNAME());
END_IF

IF NOT _DispatchValid() THEN
	RETURN;
ELSE
	_BuildCommandStringNoArgs();
	
	IF iBufferSend <> 0 AND __QUERYINTERFACE(iBufferSend, testIBufferSend) THEN
		iBufferSend.AddObject(RefObject := ZaberCommand);
	END_IF
END_IF
END_METHOD

METHOD set_system_access
IF ZaberStatus.ComponentStatus.iLastCommand <> 0 THEN
	ZaberStatus.ComponentStatus.iLastCommand.P_CommandStatus.LastCommandMessage := Base.F_GetLastWordInString(__POUNAME());
END_IF

IF NOT _DispatchValid() THEN
	RETURN;
ELSE
	_BuildCommandStringNoArgs();
	
	IF iBufferSend <> 0 AND __QUERYINTERFACE(iBufferSend, testIBufferSend) THEN
		iBufferSend.AddObject(RefObject := ZaberCommand);
	END_IF
END_IF
END_METHOD

METHOD set_system_axiscount
IF ZaberStatus.ComponentStatus.iLastCommand <> 0 THEN
	ZaberStatus.ComponentStatus.iLastCommand.P_CommandStatus.LastCommandMessage := Base.F_GetLastWordInString(__POUNAME());
END_IF

IF NOT _DispatchValid() THEN
	RETURN;
ELSE
	_BuildCommandStringNoArgs();
	
	IF iBufferSend <> 0 AND __QUERYINTERFACE(iBufferSend, testIBufferSend) THEN
		iBufferSend.AddObject(RefObject := ZaberCommand);
	END_IF
END_IF
END_METHOD

METHOD set_system_led_enable
IF ZaberStatus.ComponentStatus.iLastCommand <> 0 THEN
	ZaberStatus.ComponentStatus.iLastCommand.P_CommandStatus.LastCommandMessage := Base.F_GetLastWordInString(__POUNAME());
END_IF

IF NOT _DispatchValid() THEN
	RETURN;
ELSE
	_BuildCommandStringNoArgs();
	
	IF iBufferSend <> 0 AND __QUERYINTERFACE(iBufferSend, testIBufferSend) THEN
		iBufferSend.AddObject(RefObject := ZaberCommand);
	END_IF
END_IF
END_METHOD

METHOD set_system_serial
IF ZaberStatus.ComponentStatus.iLastCommand <> 0 THEN
	ZaberStatus.ComponentStatus.iLastCommand.P_CommandStatus.LastCommandMessage := Base.F_GetLastWordInString(__POUNAME());
END_IF

IF NOT _DispatchValid() THEN
	RETURN;
ELSE
	_BuildCommandStringNoArgs();
	
	IF iBufferSend <> 0 AND __QUERYINTERFACE(iBufferSend, testIBufferSend) THEN
		iBufferSend.AddObject(RefObject := ZaberCommand);
	END_IF
END_IF
END_METHOD

METHOD set_system_temperature
IF ZaberStatus.ComponentStatus.iLastCommand <> 0 THEN
	ZaberStatus.ComponentStatus.iLastCommand.P_CommandStatus.LastCommandMessage := Base.F_GetLastWordInString(__POUNAME());
END_IF

IF NOT _DispatchValid() THEN
	RETURN;
ELSE
	_BuildCommandStringNoArgs();
	
	IF iBufferSend <> 0 AND __QUERYINTERFACE(iBufferSend, testIBufferSend) THEN
		iBufferSend.AddObject(RefObject := ZaberCommand);
	END_IF
END_IF
END_METHOD

METHOD set_system_uptime
IF ZaberStatus.ComponentStatus.iLastCommand <> 0 THEN
	ZaberStatus.ComponentStatus.iLastCommand.P_CommandStatus.LastCommandMessage := Base.F_GetLastWordInString(__POUNAME());
END_IF

IF NOT _DispatchValid() THEN
	RETURN;
ELSE
	_BuildCommandStringNoArgs();
	
	IF iBufferSend <> 0 AND __QUERYINTERFACE(iBufferSend, testIBufferSend) THEN
		iBufferSend.AddObject(RefObject := ZaberCommand);
	END_IF
END_IF
END_METHOD

METHOD set_system_voltage
IF ZaberStatus.ComponentStatus.iLastCommand <> 0 THEN
	ZaberStatus.ComponentStatus.iLastCommand.P_CommandStatus.LastCommandMessage := Base.F_GetLastWordInString(__POUNAME());
END_IF

IF NOT _DispatchValid() THEN
	RETURN;
ELSE
	_BuildCommandStringNoArgs();
	
	IF iBufferSend <> 0 AND __QUERYINTERFACE(iBufferSend, testIBufferSend) THEN
		iBufferSend.AddObject(RefObject := ZaberCommand);
	END_IF
END_IF
END_METHOD

METHOD set_trigger_numactions
IF ZaberStatus.ComponentStatus.iLastCommand <> 0 THEN
	ZaberStatus.ComponentStatus.iLastCommand.P_CommandStatus.LastCommandMessage := Base.F_GetLastWordInString(__POUNAME());
END_IF

IF NOT _DispatchValid() THEN
	RETURN;
ELSE
	_BuildCommandStringNoArgs();
	
	IF iBufferSend <> 0 AND __QUERYINTERFACE(iBufferSend, testIBufferSend) THEN
		iBufferSend.AddObject(RefObject := ZaberCommand);
	END_IF
END_IF
END_METHOD

METHOD set_trigger_numtriggers
IF ZaberStatus.ComponentStatus.iLastCommand <> 0 THEN
	ZaberStatus.ComponentStatus.iLastCommand.P_CommandStatus.LastCommandMessage := Base.F_GetLastWordInString(__POUNAME());
END_IF

IF NOT _DispatchValid() THEN
	RETURN;
ELSE
	_BuildCommandStringNoArgs();
	
	IF iBufferSend <> 0 AND __QUERYINTERFACE(iBufferSend, testIBufferSend) THEN
		iBufferSend.AddObject(RefObject := ZaberCommand);
	END_IF
END_IF
END_METHOD

METHOD set_user_data_0
IF ZaberStatus.ComponentStatus.iLastCommand <> 0 THEN
	ZaberStatus.ComponentStatus.iLastCommand.P_CommandStatus.LastCommandMessage := Base.F_GetLastWordInString(__POUNAME());
END_IF

IF NOT _DispatchValid() THEN
	RETURN;
ELSE
	_BuildCommandStringNoArgs();
	
	IF iBufferSend <> 0 AND __QUERYINTERFACE(iBufferSend, testIBufferSend) THEN
		iBufferSend.AddObject(RefObject := ZaberCommand);
	END_IF
END_IF
END_METHOD

METHOD set_user_data_1
IF ZaberStatus.ComponentStatus.iLastCommand <> 0 THEN
	ZaberStatus.ComponentStatus.iLastCommand.P_CommandStatus.LastCommandMessage := Base.F_GetLastWordInString(__POUNAME());
END_IF

IF NOT _DispatchValid() THEN
	RETURN;
ELSE
	_BuildCommandStringNoArgs();
	
	IF iBufferSend <> 0 AND __QUERYINTERFACE(iBufferSend, testIBufferSend) THEN
		iBufferSend.AddObject(RefObject := ZaberCommand);
	END_IF
END_IF
END_METHOD

METHOD set_user_data_10
IF ZaberStatus.ComponentStatus.iLastCommand <> 0 THEN
	ZaberStatus.ComponentStatus.iLastCommand.P_CommandStatus.LastCommandMessage := Base.F_GetLastWordInString(__POUNAME());
END_IF

IF NOT _DispatchValid() THEN
	RETURN;
ELSE
	_BuildCommandStringNoArgs();
	
	IF iBufferSend <> 0 AND __QUERYINTERFACE(iBufferSend, testIBufferSend) THEN
		iBufferSend.AddObject(RefObject := ZaberCommand);
	END_IF
END_IF
END_METHOD

METHOD set_user_data_11
IF ZaberStatus.ComponentStatus.iLastCommand <> 0 THEN
	ZaberStatus.ComponentStatus.iLastCommand.P_CommandStatus.LastCommandMessage := Base.F_GetLastWordInString(__POUNAME());
END_IF

IF NOT _DispatchValid() THEN
	RETURN;
ELSE
	_BuildCommandStringNoArgs();
	
	IF iBufferSend <> 0 AND __QUERYINTERFACE(iBufferSend, testIBufferSend) THEN
		iBufferSend.AddObject(RefObject := ZaberCommand);
	END_IF
END_IF
END_METHOD

METHOD set_user_data_12
IF ZaberStatus.ComponentStatus.iLastCommand <> 0 THEN
	ZaberStatus.ComponentStatus.iLastCommand.P_CommandStatus.LastCommandMessage := Base.F_GetLastWordInString(__POUNAME());
END_IF

IF NOT _DispatchValid() THEN
	RETURN;
ELSE
	_BuildCommandStringNoArgs();
	
	IF iBufferSend <> 0 AND __QUERYINTERFACE(iBufferSend, testIBufferSend) THEN
		iBufferSend.AddObject(RefObject := ZaberCommand);
	END_IF
END_IF
END_METHOD

METHOD set_user_data_13
IF ZaberStatus.ComponentStatus.iLastCommand <> 0 THEN
	ZaberStatus.ComponentStatus.iLastCommand.P_CommandStatus.LastCommandMessage := Base.F_GetLastWordInString(__POUNAME());
END_IF

IF NOT _DispatchValid() THEN
	RETURN;
ELSE
	_BuildCommandStringNoArgs();
	
	IF iBufferSend <> 0 AND __QUERYINTERFACE(iBufferSend, testIBufferSend) THEN
		iBufferSend.AddObject(RefObject := ZaberCommand);
	END_IF
END_IF
END_METHOD

METHOD set_user_data_14
IF ZaberStatus.ComponentStatus.iLastCommand <> 0 THEN
	ZaberStatus.ComponentStatus.iLastCommand.P_CommandStatus.LastCommandMessage := Base.F_GetLastWordInString(__POUNAME());
END_IF

IF NOT _DispatchValid() THEN
	RETURN;
ELSE
	_BuildCommandStringNoArgs();
	
	IF iBufferSend <> 0 AND __QUERYINTERFACE(iBufferSend, testIBufferSend) THEN
		iBufferSend.AddObject(RefObject := ZaberCommand);
	END_IF
END_IF
END_METHOD

METHOD set_user_data_15
IF ZaberStatus.ComponentStatus.iLastCommand <> 0 THEN
	ZaberStatus.ComponentStatus.iLastCommand.P_CommandStatus.LastCommandMessage := Base.F_GetLastWordInString(__POUNAME());
END_IF

IF NOT _DispatchValid() THEN
	RETURN;
ELSE
	_BuildCommandStringNoArgs();
	
	IF iBufferSend <> 0 AND __QUERYINTERFACE(iBufferSend, testIBufferSend) THEN
		iBufferSend.AddObject(RefObject := ZaberCommand);
	END_IF
END_IF
END_METHOD

METHOD set_user_data_2
IF ZaberStatus.ComponentStatus.iLastCommand <> 0 THEN
	ZaberStatus.ComponentStatus.iLastCommand.P_CommandStatus.LastCommandMessage := Base.F_GetLastWordInString(__POUNAME());
END_IF

IF NOT _DispatchValid() THEN
	RETURN;
ELSE
	_BuildCommandStringNoArgs();
	
	IF iBufferSend <> 0 AND __QUERYINTERFACE(iBufferSend, testIBufferSend) THEN
		iBufferSend.AddObject(RefObject := ZaberCommand);
	END_IF
END_IF
END_METHOD

METHOD set_user_data_3
IF ZaberStatus.ComponentStatus.iLastCommand <> 0 THEN
	ZaberStatus.ComponentStatus.iLastCommand.P_CommandStatus.LastCommandMessage := Base.F_GetLastWordInString(__POUNAME());
END_IF

IF NOT _DispatchValid() THEN
	RETURN;
ELSE
	_BuildCommandStringNoArgs();
	
	IF iBufferSend <> 0 AND __QUERYINTERFACE(iBufferSend, testIBufferSend) THEN
		iBufferSend.AddObject(RefObject := ZaberCommand);
	END_IF
END_IF
END_METHOD

METHOD set_user_data_4
IF ZaberStatus.ComponentStatus.iLastCommand <> 0 THEN
	ZaberStatus.ComponentStatus.iLastCommand.P_CommandStatus.LastCommandMessage := Base.F_GetLastWordInString(__POUNAME());
END_IF

IF NOT _DispatchValid() THEN
	RETURN;
ELSE
	_BuildCommandStringNoArgs();
	
	IF iBufferSend <> 0 AND __QUERYINTERFACE(iBufferSend, testIBufferSend) THEN
		iBufferSend.AddObject(RefObject := ZaberCommand);
	END_IF
END_IF
END_METHOD

METHOD set_user_data_5
IF ZaberStatus.ComponentStatus.iLastCommand <> 0 THEN
	ZaberStatus.ComponentStatus.iLastCommand.P_CommandStatus.LastCommandMessage := Base.F_GetLastWordInString(__POUNAME());
END_IF

IF NOT _DispatchValid() THEN
	RETURN;
ELSE
	_BuildCommandStringNoArgs();
	
	IF iBufferSend <> 0 AND __QUERYINTERFACE(iBufferSend, testIBufferSend) THEN
		iBufferSend.AddObject(RefObject := ZaberCommand);
	END_IF
END_IF
END_METHOD

METHOD set_user_data_6
IF ZaberStatus.ComponentStatus.iLastCommand <> 0 THEN
	ZaberStatus.ComponentStatus.iLastCommand.P_CommandStatus.LastCommandMessage := Base.F_GetLastWordInString(__POUNAME());
END_IF

IF NOT _DispatchValid() THEN
	RETURN;
ELSE
	_BuildCommandStringNoArgs();
	
	IF iBufferSend <> 0 AND __QUERYINTERFACE(iBufferSend, testIBufferSend) THEN
		iBufferSend.AddObject(RefObject := ZaberCommand);
	END_IF
END_IF
END_METHOD

METHOD set_user_data_7
IF ZaberStatus.ComponentStatus.iLastCommand <> 0 THEN
	ZaberStatus.ComponentStatus.iLastCommand.P_CommandStatus.LastCommandMessage := Base.F_GetLastWordInString(__POUNAME());
END_IF

IF NOT _DispatchValid() THEN
	RETURN;
ELSE
	_BuildCommandStringNoArgs();
	
	IF iBufferSend <> 0 AND __QUERYINTERFACE(iBufferSend, testIBufferSend) THEN
		iBufferSend.AddObject(RefObject := ZaberCommand);
	END_IF
END_IF
END_METHOD

METHOD set_user_data_8
IF ZaberStatus.ComponentStatus.iLastCommand <> 0 THEN
	ZaberStatus.ComponentStatus.iLastCommand.P_CommandStatus.LastCommandMessage := Base.F_GetLastWordInString(__POUNAME());
END_IF

IF NOT _DispatchValid() THEN
	RETURN;
ELSE
	_BuildCommandStringNoArgs();
	
	IF iBufferSend <> 0 AND __QUERYINTERFACE(iBufferSend, testIBufferSend) THEN
		iBufferSend.AddObject(RefObject := ZaberCommand);
	END_IF
END_IF
END_METHOD

METHOD set_user_data_9
IF ZaberStatus.ComponentStatus.iLastCommand <> 0 THEN
	ZaberStatus.ComponentStatus.iLastCommand.P_CommandStatus.LastCommandMessage := Base.F_GetLastWordInString(__POUNAME());
END_IF

IF NOT _DispatchValid() THEN
	RETURN;
ELSE
	_BuildCommandStringNoArgs();
	
	IF iBufferSend <> 0 AND __QUERYINTERFACE(iBufferSend, testIBufferSend) THEN
		iBufferSend.AddObject(RefObject := ZaberCommand);
	END_IF
END_IF
END_METHOD

METHOD set_user_vdata_0
IF ZaberStatus.ComponentStatus.iLastCommand <> 0 THEN
	ZaberStatus.ComponentStatus.iLastCommand.P_CommandStatus.LastCommandMessage := Base.F_GetLastWordInString(__POUNAME());
END_IF

IF NOT _DispatchValid() THEN
	RETURN;
ELSE
	_BuildCommandStringNoArgs();
	
	IF iBufferSend <> 0 AND __QUERYINTERFACE(iBufferSend, testIBufferSend) THEN
		iBufferSend.AddObject(RefObject := ZaberCommand);
	END_IF
END_IF
END_METHOD

METHOD set_user_vdata_1
IF ZaberStatus.ComponentStatus.iLastCommand <> 0 THEN
	ZaberStatus.ComponentStatus.iLastCommand.P_CommandStatus.LastCommandMessage := Base.F_GetLastWordInString(__POUNAME());
END_IF

IF NOT _DispatchValid() THEN
	RETURN;
ELSE
	_BuildCommandStringNoArgs();
	
	IF iBufferSend <> 0 AND __QUERYINTERFACE(iBufferSend, testIBufferSend) THEN
		iBufferSend.AddObject(RefObject := ZaberCommand);
	END_IF
END_IF
END_METHOD

METHOD set_user_vdata_2
IF ZaberStatus.ComponentStatus.iLastCommand <> 0 THEN
	ZaberStatus.ComponentStatus.iLastCommand.P_CommandStatus.LastCommandMessage := Base.F_GetLastWordInString(__POUNAME());
END_IF

